// ---- POUs/Target/FB_PID.TcPOU
FUNCTION_BLOCK FB_PID
VAR_INPUT
	fSetpointValue: LREAL:=0;
	fActualValue :LREAL :=0;
	fFF:LREAL:=0;
	fKp: LREAL:=0;
	fKi: LREAL:=0;
	fKd: LREAL:=0;
	fKff: LREAL:=0;
	fIOutputMin: LREAL:=0;
	fIOutputMax: LREAL:=0;
	fOutputMin:LREAL:=0;
	fOutputMax:LREAL:=0;
	bReset:BOOL:=FALSE;
END_VAR
VAR_OUTPUT
	fCtrlOutput: LREAL;
END_VAR
VAR
	fOutputFF:LREAL:=0;
    fOutputP:LREAL:=0;
	fOutputI:LREAL:=0;
	fOutputD:LREAL:=0;
	fError:LREAL:=0;
	fErrorOld:LREAL:=0;
END_VAR

// Function: Simple PID controller with FF and limits for integral..
// Custom implementation needed since integral high and low limits are 
// needed in order to prvent integral windup.
// Author: Anders Sandström 20200115
 
IF bReset THEN
  fOutputP:=0;
  fOutputI:=0;
  fOutputD:=0;
  fFF:=0;
  fCtrlOutput:=0;
  RETURN;
END_IF

fErrorOld := fError;
fError    := fActualValue-fSetpointValue;

fOutputFF := fFF*fKff;         
fOutputP  := fKp*fError;
fOutputI  := fOutputI + fKi* fError;
// Prevent integral windup
IF fOutputI > fIOutputMax THEN
  fOutputI := fIOutputMax;
ELSIF fOutputI < fIOutputMin THEN
  fOutputI := fIOutputMin; 
END_IF

fOutputD  :=  (fError-fErrorOld)*fKd;

fCtrlOutput := fOutputP + fOutputI + fOutputD + fOutputFF;
IF fCtrlOutput < fOutputMin THEN
  fCtrlOutput := fOutputMin;
ELSIF fCtrlOutput > fOutputMax THEN
  fCtrlOutput := fOutputMax;
END_IF

END_FUNCTION_BLOCK

// ---- POUs/Target/FB_PWM.TcPOU
FUNCTION_BLOCK FB_PWM
VAR_INPUT
	En: BOOL;
	bEnable: BOOL;                  // Enable PWM alg
	iBlockSampleTimeMicroS: DINT;   // How often this block is called 
	iProcessSampleTimeMicroS: DINT; // Pwm cycle time. iProcessSampleTimeMicroS >> iBlockSampleTimeMicroS to get a good PWM resolution
 	iDecimalPoint: INT;             // At which decimal should teh pwm take place
	fInput: LREAL;                  // Input process value (that will be PWM:ed) 
	// PWM type:
	// Optimized: The low and high values are as ebenly distibuted in time as possible
	// Simple:    Either the low or high values are output first then the other (depending on bPromoteHigh bit)
	ePwmType:E_PWM_TYPE:=E_PWM_TYPE.OPTIMIZED;  
	bPromoteHigh:BOOL:=TRUE; // Only used in simple mode.
END_VAR
VAR_OUTPUT
	EnO: BOOL;
	fOutput: LREAL;
	fOutputError:LREAL:=0;  // Esitmated error of the PWM alg.
END_VAR
VAR
	iNumCycles: DINT;
	iBase: DINT;
	fDecimals: LREAL;
	i: INT;
	iDecimalGain: DINT;
	fOutputHigh: LREAL;
	iHighCycles: DINT;
	iLowCycles: DINT;
	fOutputLow: LREAL;
	iCycleCounter: DINT;
	iLowCounter: INT;
	iHighCounter: INT;
	fActualPWM: LREAL;
	fSetpointPWM: LREAL;
	fInputOld:LREAL:=0;
END_VAR

// Function: PWM block to be used to enhance resolution of signals
//
// Usefull for instance when a ethercat slave communicates with ints and you need 
// higher precision than the int provides. The desired input value are then PWM so that the
// average over processSampleTime is as close as possile to the desired value.
// Block can execute in three different modes:
//   OPTIMIZED: The low and high values are as evently as possible distributed over time
//   SIMPLE:    All high or low values are output first then the other (depending on bPromoteHigh bit)
//   NONE:      Output is same as input (no PWM)
//
// Note: Average resolution will be higher on the cost of sample rate
// Note: Error of PWM alg can be seen in fOutputError
//
// Example: fInput = 23.33333333, iDecimalpoint=3  ==>
//            fOutput will be pulse width modulated with the two discrete values: 23.333 and 23.334
//            in 33% of iProcessSampleTimeMicroS fOutput will be 23.333 and
//            in 67% of iProcessSampleTimeMicroS fOutput will be 23.334
//
// Author: Anders Sandström 2018
//
IF bEnable THEN
  IF(fInput<>fInputOld) THEN // New input value
    iNumCycles:=iProcessSampleTimeMicroS/iBlockSampleTimeMicroS; //71 if 71ms and 1ms
	iDecimalGain:=1;
	FOR i:=1 TO iDecimalPoint DO
      iDecimalGain:=iDecimalGain*10; //10000 if iDecimalpoint is 4
	END_FOR
	iBase:=TRUNC(fInput*iDecimalGain); //=900004 if fOverride=90.00045
    fDecimals:=fInput*iDecimalGain-iBase; //=0.5 if fOverride=90.00045
	iHighCycles:=LREAL_TO_INT(iNumCycles*fDecimals);
    iLowCycles:=iNumCycles-iHighCycles;
    fOutputLow:=DINT_TO_LREAL(iBase)/iDecimalGain; //90.0004
    fOutputHigh:=DINT_TO_LREAL(iBase+1)/iDecimalGain; //90.0005
	iCycleCounter:=0;
	iLowCounter:=0;
	iHighCounter:=0;
	fOutputError:=(fDecimals-DINT_TO_LREAL(iHighCycles)/DINT_TO_LREAL(iNumCycles))/iDecimalGain;
	fSetpointPWM:=DINT_TO_LREAL(iHighCycles)/DINT_TO_LREAL(iLowCycles+iHighCycles);
    END_IF

    IF iCycleCounter > iNumCycles THEN
	  iCycleCounter:=0;
	  iLowCounter:=0;
	  iHighCounter:=0;	
    END_IF
    iCycleCounter:=iCycleCounter+1;
	
  CASE ePwmType OF
	E_PWM_TYPE.OPTIMIZED:  // Distribute low and high evenly in time
       IF iLowCycles > 0 THEN
	     IF iHighCycles > 0 THEN
	       //Both high and low should be output during the period
	       IF iLowCounter = 0 THEN
		     fOutput:=fOutputLow;
		     iLowCounter:=iLowCounter+1;
	       ELSE
	         IF iHighCounter = 0 THEN
		       fOutput:=fOutputHigh;
		       iHighCounter:=iHighCounter+1;
	         ELSE //both counters is atleast 1
		       fActualPWM:= DINT_TO_LREAL(iHighCounter)/DINT_TO_LREAL(iLowCounter+iHighCounter);
		       IF fActualPWM>fSetpointPWM THEN
		         fOutput:=fOutputLow;
		         iLowCounter:=iLowCounter+1;
		       ELSE
                 fOutput:=fOutputHigh;
		         iHighCounter:=iHighCounter+1;
		       END_IF				
	        END_IF				
	      END_IF
        ELSE		
	      fOutput:=fOutputLow;
	      iLowCounter:=iLowCounter+1;
        END_IF
      ELSE
        fOutput:=fOutputHigh;
	    iHighCounter:=iHighCounter+1;
      END_IF
	  
    E_PWM_TYPE.SIMPLE:  // Take all low or high first then the other
	  IF bPromoteHigh THEN  // All high first
        IF iHighCounter < iHighCycles THEN
          iHighCounter:=iHighCounter+1;
		  fOutput:=fOutputHigh;
		ELSE
		  iLowCounter:=iLowCounter+1;
		  fOutput:=fOutputLow;
        END_IF
	  ELSE                  // All low first
        IF iLowCounter < iLowCycles THEN
          iLowCounter:=iLowCounter+1;
		  fOutput:=fOutputLow;
		ELSE
		  iHighCounter:=iHighCounter+1;
		  fOutput:=fOutputHigh;
        END_IF
		  
	  END_IF
	E_PWM_TYPE.NONE:    // Output same as input
	  fOutput:=fInput;
	  iCycleCounter:=0;
	  iLowCounter:=0;
	  iHighCounter:=0;	
	END_CASE
    
ELSE	
	fOutput:=fInput;	
END_IF
fInputOld:=fInput;

END_FUNCTION_BLOCK

// ---- POUs/Target/FB_RampVelo.TcPOU
FUNCTION_BLOCK FB_RampVelo
VAR_INPUT
	bExecute:BOOL;
	fVelSetIn:LREAL:=0;
	iBlockSampleTimeMicroS:INT:=10000;
	fVelActIn:LREAL:=0;
END_VAR
VAR_IN_OUT
    fVelSetOut:LREAL:=0;
END_VAR
VAR
  fChangePerCycle:LREAL:=0;
  fCurrAcc:LREAL:=0;
  fAccX1:LREAL:=0.8;
  fAccX2:LREAL:=0.99;
  fAccY1:LREAL:=GVL_Parameters.fAccDefaultVel;
  fAccY2:LREAL:=GVL_Parameters.fAccDefaultVel*0.1;
  fAccK:LREAL:=0;
  fAccM:LREAL:=0;
  x:LREAL:=0;
  bExecuteOld:BOOL:=FALSE;
  fActVeloOld:LREAL:=0;  // Used for extra sanity check of velo
END_VAR

// Function: Ramp velocity with a defined acceleration.
// Accelerartion is ramped down when approaching velocity setpoint in order to reduce
// overshoot and oscillations..
// Author: Anders Sandström 20200114

IF NOT bExecute OR ABS(fVelSetIn) > GVL_Parameters.fMaximumSPeedSPRpm THEN
  fVelSetOut:=0;
  bExecuteOld:=bExecute;
  fActVeloOld:=fVelActIn;
  RETURN;
END_IF;

// Start at current velocity if retreigger (avoid go to zero)
IF NOT bExecuteOld AND bExecute THEN
  // Sanity check of the actual velocity
  IF fVelActIn > -GVL_Parameters.fMaximumSPeedRpm AND 
	 fVelActIn < GVL_Parameters.fMaximumSPeedRpm AND 
	 fActVeloOld > -GVL_Parameters.fMaximumSPeedRpm AND 
	 fActVeloOld < GVL_Parameters.fMaximumSPeedRpm THEN
	fVelSetOut:=(fVelActIn+fActVeloOld)/2;  //Set to average of two cycles
    
	//Ensure minimum velo setpoint positive  to allow smooth start (with high ff tourqe at start)
	IF fVelSetIn > 0 AND ABS(fVelSetOut) < GVL_Parameters.fMinVelSetpointAbsRpm THEN
		fVelSetOut:=GVL_Parameters.fMinVelSetpointAbsRpm;
	END_IF
	//Ensure minimum velo setpoint negative to allow smooth start (with high ff tourqu at start)
	IF fVelSetIn < 0 AND ABS(fVelSetOut) < GVL_Parameters.fMinVelSetpointAbsRpm THEN
		fVelSetOut:=-GVL_Parameters.fMinVelSetpointAbsRpm;
	END_IF
  ELSE
    fVelSetOut:=0;
  END_IF  
END_IF
bExecuteOld:=bExecute;
fActVeloOld:=fVelActIn;

IF fVelSetOut=fVelSetIn THEN
  fVelSetOut:=fVelSetIn;
  RETURN;
END_IF;

//Reduce overshoot by lowering acc when closing in on setpoint (linear)
//           Acceleration [rpm/s^2]
//                 ^
//  y1=defAcc     -|-----------------\
//                 |                  \  
//                 |                   \
//                 |                    \ 
//                 |                     \
//  y2=defAcc*0.1 -|                      \-----------------
//                 |--------------------------------------------> fSetOut/fSetIn []
//                                 x1=0.8 x2=1.0 

fAccK:=(fAccY2-fAccY1)/(fAccX2-fAccX1);
fAccM:= fAccY1-fAccK*fAccX1;
IF fVelSetIn<>0 THEN
  x:=fVelSetOut/fVelSetIn;
ELSE
  x:=1.0;
END_IF
// try linear ramp down off acceleration from 0.8*velsetin to velset in (from defacc to 0.1* defacc)
fCurrAcc:=GVL_Parameters.fAccDefaultVel;
IF fVelSetIn > fVelSetOut THEN 
  IF x > fAccX1 AND x <= fAccX2 AND fVelSetOut<fVelSetIn THEN
    fCurrAcc:=fAccK*fVelSetOut/fVelSetIn+fAccM;
  ELSIF x >= fAccX2 THEN
    fCurrAcc:=GVL_Parameters.fAccDefaultVel*0.1;
  END_IF
END_IF

// Change per execution
fChangePerCycle:=fCurrAcc/(1E6/iBlockSampleTimeMicroS);

// Ramp finished
IF ABS(fVelSetIn-fVelSetOut)<fChangePerCycle THEN
  fVelSetOut:=fVelSetIn;
  RETURN;
END_IF

//Acc
IF fVelSetIn > fVelSetOut THEN             // Acc
  fVelSetOut:=fVelSetOut+fChangePerCycle;
ELSIF fVelSetIn < fVelSetOut THEN          // Dec
  fVelSetOut:=fVelSetOut-fChangePerCycle;
END_IF

END_FUNCTION_BLOCK

// ---- POUs/Target/FB_ModeVelo.TcPOU
FUNCTION_BLOCK FB_ModeVelo
VAR_INPUT
	bExecute:BOOL;
	bReset: BOOL;
	fVelSet:LREAL:=0;
	stStatus: ST_INDRADRIVE_AXIS_STATUS;
END_VAR
VAR_OUTPUT
	fSpeedSetpoint:LREAL:=0;
	bError: BOOL;
	nErrorId: UDINT;
	sErrorStr: STRING:=GVL_ErrorCodes.nErrorCodeOKStr;
END_VAR
VAR_IN_OUT
	stCommands: ST_INDRADRIVE_AXIS_COMMAND;
END_VAR

// Function: Constant velocity of target main  motor
// Control will be performed by the drive.
// Author: Anders Sandström 2018

stCommands.eMotionMode :=e_Motion_mode.eJogPositive;
stCommands.eOperationMode:=e_Operation_mode_no.eSecondaryOpMode2;
IF bExecute THEN
	fSpeedSetpoint:=fVelSet;
ELSE
	fSpeedSetpoint:=0;
END_IF
stCommands.fCommandVelocity:=0; // Other mode

END_FUNCTION_BLOCK

// ---- POUs/Target/FB_ModePos.TcPOU
FUNCTION_BLOCK FB_ModePos
VAR_INPUT
	bExecute:BOOL;
	bReset: BOOL;
	fVelSet:LREAL:=0;
	fPosSet:LREAL:=0;
	fRefOffset:LREAL:=0;  //Offset from homing
	stStatus: ST_INDRADRIVE_AXIS_STATUS;
END_VAR
VAR_OUTPUT
	bError: BOOL;
	nErrorId: UDINT;
	sErrorStr: STRING:=GVL_ErrorCodes.nErrorCodeOKStr;
END_VAR
VAR_IN_OUT
	stCommands: ST_INDRADRIVE_AXIS_COMMAND;
END_VAR
VAR
	fActPos:LREAL:=0;
    bExecuteOld:BOOL:=FALSE;
    //fPosSetTemp:LREAL:=0;
	fDistToTarget:LREAL:=0;
	//fDistToTrajSet:LREAL:=0;
	bVeloMode:BOOL:=FALSE;
END_VAR

// Function: Absolute positioning of target main  motor
// Actual positioning will be performed by the drive.
// Author: Anders Sandström 2018

stCommands.eMotionMode :=e_Motion_mode.ePositioning;
stCommands.eOperationMode:=e_Operation_mode_no.ePrimaryOpMode;
//stCommands.eOperationMode:=e_Operation_mode_no.eSecondaryOpMode3;

fActPos:=stStatus.fActualPosition-fRefOffset;
IF fActPos > 360 THEN
  fActPos:=fActPos-360;	
END_IF
IF fActPos < 0 THEN
  fActPos:=fActPos+360;	
END_IF

fDistToTarget:=FC_DistMod(fPosFrom:=fActPos,fPosTo:=fPosSet,fModRange:=360);
IF bExecute AND  NOT bExecuteOld THEN
  IF ABS(fDistToTarget) > 30 THEN   
    bVeloMode:=TRUE;
  ELSE
    bVeloMode:=FALSE;	 
  END_IF
END_IF

IF NOT bExecute THEN
  bVeloMode:=FALSE;
END_IF;	 
IF bExecute THEN
  IF bVeloMode THEN
	IF fDistToTarget> 0 THEN
	  stCommands.fVelocityCommandValue:=fVelSet;
	  IF fDistToTarget>0 THEN
	    stCommands.eMotionMode :=e_Motion_mode.eJogPositive;
	  ELSE
		 stCommands.eMotionMode :=e_Motion_mode.eJogNegative;
	  END_IF
      stCommands.eOperationMode:=e_Operation_mode_no.eSecondaryOpMode2;
	END_IF
	IF ABS(fDistToTarget) < 30 THEN 
		stCommands.fVelocityCommandValue:=0;
		IF stStatus.fActualVelocity <  fVelSet THEN
			bVeloMode:=FALSE;
		END_IF
	END_IF
  ELSE   // positioning
      stCommands.fCommandPosition:=fPosSet + fRefOffset;
      IF stCommands.fCommandPosition > 360 THEN
        stCommands.fCommandPosition:=stCommands.fCommandPosition-360;	
      END_IF
      IF stCommands.fCommandPosition < 0 THEN
         stCommands.fCommandPosition:=stCommands.fCommandPosition+360;	
      END_IF
      stCommands.fCommandVelocity:=fVelSet;
	  stCommands.eMotionMode :=e_Motion_mode.ePositioning;
      stCommands.eOperationMode:=e_Operation_mode_no.ePrimaryOpMode;
	  stCommands.fVelocityCommandValue:=0;
  END_IF
ELSE  
  stCommands.fCommandVelocity:=0;
  stCommands.fVelocityCommandValue:=0;
END_IF


//fDistToTrajSet:=FC_DistMod(fPosFrom:=fActPos,fPosTo:=fPosSetTemp,fModRange:=360);


(*IF ABS(fDistToTrajSet) < GVL_Parameters.fReachedTol THEN
  IF fDistToTarget > 0 THEN  // Increase traj setpoint with one step
	  fPosSetTemp:= fPosSetTemp + GVL_Parameters.fPosStep;
  ELSE
	  fPosSetTemp:= fPosSetTemp - GVL_Parameters.fPosStep;
  END_IF
END_IF

IF ABS(fDistToTarget) < GVL_Parameters.fPosStep THEN
   fPosSetTemp:=fPosSet;
END_IF

IF bExecute THEN
  stCommands.fCommandPosition:=fPosSetTemp + fRefOffset;
  IF stCommands.fCommandPosition > 360 THEN
    stCommands.fCommandPosition:=stCommands.fCommandPosition-360;	
  END_IF
  IF stCommands.fCommandPosition < 0 THEN
    stCommands.fCommandPosition:=stCommands.fCommandPosition+360;	
  END_IF
  stCommands.fCommandVelocity:=fVelSet;
ELSE
  stCommands.fCommandPosition:=stStatus.fActualPosition;
  stCommands.fCommandVelocity:=0;
END_IF*)


//stCommands.fVelocityCommandValue:=0;  //Used for other mode
bExecuteOld:=bExecute;

END_FUNCTION_BLOCK

// ---- POUs/Target/FB_ModeHome.TcPOU
FUNCTION_BLOCK FB_ModeHome
VAR_INPUT
	bExecute           : BOOL  := FALSE;
	bReset             : BOOL  := FALSE;
	fVelSet            : LREAL := 0;
	fPosSet            : LREAL := 0;
	stStatus           : ST_INDRADRIVE_AXIS_STATUS;
END_VAR
VAR_OUTPUT
	fSpeedSetpoint     : LREAL  := 0;
	fActPositionOffset : LREAL  := 0;
	bBusy              : BOOL   := FALSE;
	bError             : BOOL   := 0;
	nErrorId           : UDINT  := 0;
	sErrorStr          : STRING := GVL_ErrorCodes.nErrorCodeOKStr;
END_VAR
VAR_IN_OUT
	stCommands : ST_INDRADRIVE_AXIS_COMMAND;
	bHomed     : BOOL;
END_VAR
VAR
  bRefMarkPosArrayConsistent : BOOL  := FALSE;
  bTriggLatchMark            : BOOL  := FALSE;
  bExecuteOld                : BOOL  := FALSE;  
  nRevCounter                : UDINT := 0;
  nCounter                   : UDINT := 0;
  nRefMarksTotCount          : UDINT := 0;
  i                          : UDINT := 0;
  fNewestRefMarkPos          : LREAL := 0;
  fActPosAtHomeStart         : LREAL := 0;
  fMarkerPositionOld         : LREAL := 0;
  fActPositionOld            : LREAL := 0;
  fRefMarkPosArray           : ARRAY[ 0 ..GVL_Parameters.nRefMarkArraySize] OF LREAL;
  eHomeState                 : E_HOME_STATE := E_HOME_STATE.IDLE;
END_VAR

// Function: Initiate homing of target main motor
// Homing procedure:
// 1. Ramp up to (95% of) homing velocity (GVL_Parameters.fHomeSpeedRpm)
// 2. Issue drive command C1400 (latch encoder mark position)
//    - Latch GVL_Parameters.nRefMarkArraySize times (revolutions).
//    - Check that one latch per rev occurs.
//    - Check that all the latched psoitions are same.
//    - If everything is OK then store the position offset in fActPositionOffset 
//    - and set the bHomed flag. 
// 3. Ramp down.
// 4. Homing procedure is finalized
//    Now the fActPositionOffset can be used to offset the position from the drive
//    bBusy is set to false.
//
// Note: Homing is here in TwinCAT since the built in homing procedure cannot be used since
//       position loop in the drive is imposible to tune. 
//       This procedure runs the motor in velocity mode which are used for all other modes 
//       and can be releatively well tuned.
//
// Author: Anders Sandström 2018
//

// Test to ref in const velo
stCommands.eMotionMode :=e_Motion_mode.eJogPositive;
stCommands.eOperationMode:=e_Operation_mode_no.eSecondaryOpMode2;
stCommands.bCmd_NCHomeEnable:=TRUE;  // not used
stCommands.fCommandVelocity:=0; // Other mode
stCommands.bCmd_GetMarkerPosition:=bTriggLatchMark;
// Clear array and start
IF NOT bExecute AND eHomeState <> E_HOME_STATE.IDLE THEN
  eHomeState:=E_HOME_STATE.RAMP_DOWN;
END_IF

IF bReset THEN
  bError    := FALSE;
  nErrorID  := 0;
  sErrorStr := GVL_ErrorCodes.nErrorCodeOKStr;	
END_IF

CASE eHomeState OF
  E_HOME_STATE.IDLE:
    bBusy:=FALSE;
    IF bExecute AND NOT bExecuteOld AND NOT bError THEN
	  // Clear buffer and reset variables on state transition
      MEMSET(ADR(fRefMarkPosArray),0,SIZEOF(fRefMarkPosArray));
	  bBusy              := TRUE;  
      bTriggLatchMark    := FALSE;
      bHomed             := FALSE;
      nRefMarksTotCount  := 0;
	  nRevCounter        := 0;
	  fSpeedSetpoint     := 0;
	  fActPosAtHomeStart := 0;
	  fActPositionOffset := 0;
	  fNewestRefMarkPos  := 0;
	  eHomeState:=E_HOME_STATE.RAMP_UP;
    END_IF

  E_HOME_STATE.RAMP_UP:
    // Wait until reached velocity (once)
	fSpeedSetpoint:=fVelSet;
	bBusy:=TRUE;
    IF stStatus.fActualVelocity/10 > 0.95 * GVL_Parameters.fHomeSpeedRpm THEN
	  fActPosAtHomeStart := stStatus.fActualPosition;
      eHomeState:=E_HOME_STATE.HOMING;
	  bTriggLatchMark := TRUE;
    END_IF
	
  E_HOME_STATE.HOMING:
    // Move new latched value to buffer (newest always on index 0)
    IF (*stStatus.bCmd_GetMarkerPositionDone*) fMarkerPositionOld <> stStatus.fMarkerPosition AND 
      stStatus.fMarkerPosition <> 0 THEN
      MEMMOVE(ADR(fRefMarkPosArray)+SIZEOF(LREAL),ADR(fRefMarkPosArray),SIZEOF(fRefMarkPosArray)-SIZEOF(LREAL));
      fRefMarkPosArray[0]:=stStatus.fMarkerPosition;
      nCounter:=0;
      nRefMarksTotCount:=nRefMarksTotCount+1;
      // Check that complete buffer have same value (same latched value for all revs)
      IF nRefMarksTotCount >= GVL_Parameters.nRefMarkArraySize THEN
        fNewestRefMarkPos:=fRefMarkPosArray[0];
        bRefMarkPosArrayConsistent := TRUE;
        FOR i:=1 TO GVL_Parameters.nRefMarkArraySize - 1 DO
	      IF bRefMarkPosArrayConsistent THEN
	        bRefMarkPosArrayConsistent := fRefMarkPosArray[i] = fNewestRefMarkPos;
	      END_IF
        END_FOR
        bHomed:=bRefMarkPosArrayConsistent;
		IF bHomed THEN
		  fActPositionOffset := fNewestRefMarkPos+GVL_Parameters.fRotPosOffsetDeg;
		  IF fActPositionOffset>360 THEN
			  fActPositionOffset:=fActPositionOffset-360;
		  END_IF
		  IF fActPositionOffset<0 THEN
			  fActPositionOffset:=360+fActPositionOffset;
		  END_IF
		  
		ELSE
		  bError:=TRUE;	
          nErrorId:=GVL_ErrorCodes.nErrorEncoderLatchMissMatch;
          sErrorStr:=GVL_ErrorCodes.sErrorEncoderLatchMissMatch; 
		END_IF
      END_IF
    END_IF

    // Wait 100 cycles to ensure communication with drive..
    IF stStatus.fMarkerPosition <> 0 AND nCounter > 100 THEN
      bTriggLatchMark:=NOT bTriggLatchMark;
      nCounter:=0;  // wait for "response"
    END_IF
    nCounter:=nCounter+1;
	
    // Count revs since start homing. Must be one latch per rev.
	IF stStatus.fActualPosition > fActPosAtHomeStart AND fActPositionOld <= fActPosAtHomeStart THEN
      nRevCounter := nRevCounter+1;
	END_IF
	
	IF nRevCounter - nRefMarksTotCount > 1 THEN
	  bError := TRUE;
	  nErrorID := GVL_ErrorCodes.nErrorEncoderLatchLost;
	  sErrorStr := GVL_ErrorCodes.sErrorEncoderLatchLost;
	  eHomeState := E_HOME_STATE.RAMP_DOWN;
	END_IF
	
	IF nRefMarksTotCount > GVL_Parameters.nRefMarkArraySize OR bError THEN
	  eHomeState := E_HOME_STATE.RAMP_DOWN;
	END_IF
	
  E_HOME_STATE.RAMP_DOWN:
    fSpeedSetpoint:=0;
	IF stStatus.bAxisStandStillStatus THEN
	  eHomeState:=E_HOME_STATE.IDLE;
	  bBusy:=FALSE;
	END_IF
	
  ELSE
	eHomeState:=E_HOME_STATE.RAMP_DOWN;	
	
END_CASE

fMarkerPositionOld:=stStatus.fMarkerPosition;
fActPositionOld := stStatus.fActualPosition;
bExecuteOld:=bExecute;

END_FUNCTION_BLOCK

// ---- POUs/Target/FB_CalcVeloFromLatch.TcPOU
FUNCTION_BLOCK FB_CalcVeloFromLatch
VAR_INPUT
    dLatchedPosition   : DINT         := 0;
	fVeloLimit         : LREAL        := 3;
END_VAR
VAR_OUTPUT
	bError             : BOOL;
	nErrorId           : UDINT;
	sErrorStr          : STRING := GVL_ErrorCodes.nErrorCodeOKStr;
	fSpeedActual       : LREAL;
END_VAR
VAR
  dLatchedPositionOld      : DINT  := 0;
  fLatchedPositionOld      : LREAL := 0;
  fDistBetweenLastPulses   : LREAL := 0;
  fLastSectorVelocity      : LREAL := 0;
  fLatchedPosition         : LREAL := 0;
  fLastSectorVelocityOld   : LREAL := 0;
 END_VAR

// Function: 
// Calc velocity from drive latched positions (latched by timing system).
// This will result in an average velocity (for each sector at nominal speed) updated at 14Hz
// Author: Anders Sandström 2022

fLatchedPositionOld:=fLatchedPosition;  // Backup old
fLatchedPosition:=DINT_TO_LREAL(dLatchedPosition)/10000.0;  // remove homing offset
IF fLatchedPosition > 360 THEN
  fLatchedPosition:=fLatchedPosition - 360;	
END_IF
IF fLatchedPosition < 0 THEN
  fLatchedPosition:=fLatchedPosition + 360;	
END_IF

// New trigger from timing system
IF (fLatchedPosition-fLatchedPositionOld)<>0 THEN
  
  fDistBetweenLastPulses:=fLatchedPosition-fLatchedPositionOld;
  // Check over/underflow
  IF (ABS(fLatchedPositionOld - fLatchedPosition) > 200 ) THEN
    IF(fLatchedPositionOld > fLatchedPosition) THEN
	  // overflow
	  fDistBetweenLastPulses:=(360 - fLatchedPositionOld+fLatchedPosition);
    ELSE
	  // underflow
	  fDistBetweenLastPulses:=  fLatchedPositionOld +  fLatchedPosition-360;  
    END_IF
  END_IF

  fLastSectorVelocity:=fDistBetweenLastPulses*GVL_Parameters.nPulseFreqHz*60/360;
  fLastSectorVelocityOld:=fLastSectorVelocity;
END_IF

dLatchedPositionOld:=dLatchedPosition;
fSpeedActual:=fLastSectorVelocity;

END_FUNCTION_BLOCK

// ---- POUs/Target/fbIndraDrive.TcPOU
FUNCTION_BLOCK fbIndraDrive
VAR_INPUT 
	AmsNetId			: AMSNETID;		// AMS Net Id of the EtherCAT Master
	AdsAddr_Port		: WORD; 		// EtherCAT address of the Drive
	stAxisCommands		: ST_INDRADRIVE_AXIS_COMMAND; 
	stDriveStatus		: ST_INDRADRIVE_IO_INPUT; 
END_VAR
VAR_OUTPUT
	stAxisStatus		: ST_INDRADRIVE_AXIS_STATUS; 
	stDriveCommands		: ST_INDRADRIVE_IO_OUTPUT; 
END_VAR
VAR
	sAmsNetId						: T_AmsNetId;
	fbReadParameter					: FB_EcSoERead;
	nS149_DataStatus				: UDINT	:= 0;
END_VAR

VAR CONSTANT
	cC1300_LimitsEnabled			: UDINT := 0;
	cC1300_LimitsDisableActivated	: UDINT := 7;
	cC1300_LimitsDisabled			: UDINT := 3;
END_VAR

//==================================================================================================
//====== FunctionBlock to manage IndraDrive status and command =====================================
//==================================================================================================

// Create the T_AmsNetId 
sAmsNetId := F_CreateAmsNetId(AmsNetId); 

(*==================================================================================================================================================
=============    STATUS FROM THE DRIVE    ==========================================================================================================
==================================================================================================================================================*)
	// Display Drive status
		// Drive parameter mode  
		stAxisStatus.bDriveInParameterMode			:= stDriveStatus.stS144_SignalStatusWord.bS424_DriveMode; 

		// Drive Operation mode number
		IF (NOT stDriveStatus.nS135_DriveStatusWord.bS135_ActualOperationMode_Bit2) AND (NOT stDriveStatus.nS135_DriveStatusWord.bS135_ActualOperationMode_Bit1) AND (NOT stDriveStatus.nS135_DriveStatusWord.bS135_ActualOperationMode_Bit0) THEN 
			stAxisStatus.eActualOperationModeNo	:= E_OPERATION_MODE_NO.ePrimaryOpMode; 
		ELSIF (NOT stDriveStatus.nS135_DriveStatusWord.bS135_ActualOperationMode_Bit2) AND (NOT stDriveStatus.nS135_DriveStatusWord.bS135_ActualOperationMode_Bit1) AND stDriveStatus.nS135_DriveStatusWord.bS135_ActualOperationMode_Bit0 THEN 
			stAxisStatus.eActualOperationModeNo	:= E_OPERATION_MODE_NO.eSecondaryOpMode1; 
		ELSIF (NOT stDriveStatus.nS135_DriveStatusWord.bS135_ActualOperationMode_Bit2) AND stDriveStatus.nS135_DriveStatusWord.bS135_ActualOperationMode_Bit1 AND (NOT stDriveStatus.nS135_DriveStatusWord.bS135_ActualOperationMode_Bit0) THEN 
			stAxisStatus.eActualOperationModeNo	:= E_OPERATION_MODE_NO.eSecondaryOpMode2; 
		ELSIF (NOT stDriveStatus.nS135_DriveStatusWord.bS135_ActualOperationMode_Bit2) AND stDriveStatus.nS135_DriveStatusWord.bS135_ActualOperationMode_Bit1 AND stDriveStatus.nS135_DriveStatusWord.bS135_ActualOperationMode_Bit0 THEN 
			stAxisStatus.eActualOperationModeNo	:= E_OPERATION_MODE_NO.eSecondaryOpMode3; 
		ELSIF stDriveStatus.nS135_DriveStatusWord.bS135_ActualOperationMode_Bit2 AND (NOT stDriveStatus.nS135_DriveStatusWord.bS135_ActualOperationMode_Bit1) AND (NOT stDriveStatus.nS135_DriveStatusWord.bS135_ActualOperationMode_Bit0) THEN 
			stAxisStatus.eActualOperationModeNo	:= E_OPERATION_MODE_NO.eSecondaryOpMode4; 
		ELSIF stDriveStatus.nS135_DriveStatusWord.bS135_ActualOperationMode_Bit2 AND (NOT stDriveStatus.nS135_DriveStatusWord.bS135_ActualOperationMode_Bit1) AND stDriveStatus.nS135_DriveStatusWord.bS135_ActualOperationMode_Bit0 THEN 
			stAxisStatus.eActualOperationModeNo	:= E_OPERATION_MODE_NO.eSecondaryOpMode5; 
		ELSIF stDriveStatus.nS135_DriveStatusWord.bS135_ActualOperationMode_Bit2 AND stDriveStatus.nS135_DriveStatusWord.bS135_ActualOperationMode_Bit1 AND (NOT stDriveStatus.nS135_DriveStatusWord.bS135_ActualOperationMode_Bit0) THEN 
			stAxisStatus.eActualOperationModeNo	:= E_OPERATION_MODE_NO.eSecondaryOpMode6; 
		ELSIF stDriveStatus.nS135_DriveStatusWord.bS135_ActualOperationMode_Bit2 AND stDriveStatus.nS135_DriveStatusWord.bS135_ActualOperationMode_Bit1 AND stDriveStatus.nS135_DriveStatusWord.bS135_ActualOperationMode_Bit0 THEN 
			stAxisStatus.eActualOperationModeNo	:= E_OPERATION_MODE_NO.eSecondaryOpMode7; 
		END_IF
		// DC Bus
		stAxisStatus.bDCBusPresent					:= (*(NOT stDriveStatus.nS135_DriveStatusWord.bS135_ReadyForOperation_Bit0) AND *) stDriveStatus.nS135_DriveStatusWord.bS135_ReadyForOperation_Bit1; 
		// Axis enabled 
		stAxisStatus.bAxisEnabled					:= stDriveStatus.nS135_DriveStatusWord.bS135_ReadyForOperation_Bit0 AND stDriveStatus.nS135_DriveStatusWord.bS135_ReadyForOperation_Bit1; 
		// Absolute position status
		stAxisStatus.bAxisHomedStatus				:= stDriveStatus.stS144_SignalStatusWord.bS403_0_AxisHomedStatus; 
		// Axis standstill status 
		stAxisStatus.bAxisStandStillStatus			:= stDriveStatus.stS144_SignalStatusWord.bS331_StandStillStatus; 
		// Axis in target position
		stAxisStatus.bAxisInTargetPosition			:= stDriveStatus.stS144_SignalStatusWord.bS437_2_CommandPositionReached;
 		// Axis in constant velocity
		stAxisStatus.bAxisConstantVelocityStatus	:= (NOT stDriveStatus.stS144_SignalStatusWord.bS331_StandStillStatus) AND (NOT stDriveStatus.stS144_SignalStatusWord.bS437_5_Acceleration) AND (NOT stDriveStatus.stS144_SignalStatusWord.bS437_6_Deceleration);
 		// Axis in Acceleration
		stAxisStatus.bAxisAccelerationStatus		:= stDriveStatus.stS144_SignalStatusWord.bS437_5_Acceleration;
 		// Axis in Deceleration
		stAxisStatus.bAxisDecelerationStatus		:= stDriveStatus.stS144_SignalStatusWord.bS437_6_Deceleration;
 		// Axis in Jog
		stAxisStatus.bAxisJogStatus					:= stDriveStatus.stS144_SignalStatusWord.bS437_12_JogMode;
		// Drive command change 
		stAxisStatus.bCommandChange					:= stDriveStatus.nS135_DriveStatusWord.bS135_CommandChange; 
		// Drive command value processing  
		stAxisStatus.bCommandValueProcessing		:= stDriveStatus.stS144_SignalStatusWord.bP115_3_StatusOfCmdValueProcessing; 
        // STO active  ch1        
        stAxisStatus.bSTOActiveCh1:= stDriveStatus.stS144_SignalStatusWord.bP106_1_STO_ch1;
		// STO active  ch2       
        stAxisStatus.bSTOActiveCh2:= stDriveStatus.stS144_SignalStatusWord.bP106_2_STO_ch2;
        // C1400 Get Marker Position
		stAxisStatus.bCmd_GetMarkerPositionDone     := stDriveStatus.stS144_SignalStatusWord.bP14_0_C1400_GetMarkerPositionDone;
		
		// Disable monitoring  
		IF 	(stAxisCommands.bCmd_DisableLimits AND (NOT stAxisStatus.bLimitsDisabled)) OR 
			((NOT stAxisCommands.bCmd_DisableLimits) AND stAxisStatus.bLimitsDisabled) THEN
				fbReadParameter(
					sNetId:= sAmsNetId, 
					nSlaveAddr:= AdsAddr_Port, 
					nIdn:= 149, 
					nElement:= 16#01, 
					nDriveNo:= 0, 
					bCommand:= FALSE, 
					pDstBuf:= ADR(nS149_DataStatus), 
					cbBufLen:= SIZEOF(nS149_DataStatus), 
					bExecute:= TRUE, 
					tTimeout:= , 
					bBusy=> , 
					bError=> , 
					nErrId=> ); 
				
				IF (NOT fbReadParameter.bBusy) AND (NOT fbReadParameter.bError) THEN 
					IF (nS149_DataStatus = cC1300_LimitsDisableActivated) OR (nS149_DataStatus = cC1300_LimitsDisabled) THEN 
						stAxisStatus.bLimitsDisabled	:= TRUE;
					ELSIF (nS149_DataStatus = cC1300_LimitsEnabled) THEN 
						stAxisStatus.bLimitsDisabled	:= FALSE;
					END_IF
					// Execute with FALSE
					fbReadParameter(bExecute:= FALSE);
				END_IF
				
				IF fbReadParameter.bError THEN 
					// Execute with FALSE
					fbReadParameter(bExecute:= FALSE);
				END_IF
		END_IF
		
		// Diagnostic message present 
		stAxisStatus.bDiagMessage					:= stDriveStatus.nS135_DriveStatusWord.bS135_Class3_Diag_Mess;  
		// Warning message present 
		stAxisStatus.bWarning						:= stDriveStatus.nS135_DriveStatusWord.bS135_Class2_Diag_Warn;  
		// Error message present 
		stAxisStatus.bError							:= stDriveStatus.nS135_DriveStatusWord.bS135_Class1_Diag_Err;  
		// Diagnostic message number 
		{attribute 'displaymode':='hexadecimal'} 
		stAxisStatus.nDiagMessage					:= stDriveStatus.nS390_DiagnosticMessageNumber;
		
		// Display motion actual values 
		// Actual position (scale by 10000) 
		stAxisStatus.fActualPosition		:= DINT_TO_LREAL(stDriveStatus.nS386_ActivePositionFeedbackValue) / 10000.0; 
		// Actual velocity (scale by 1000) 
		stAxisStatus.fActualVelocity		:= DINT_TO_LREAL(stDriveStatus.nS40_VelocityFeedbackValue) / 1000.0; 
		// Actual Torque (scale by 10) 
		stAxisStatus.fActualTorque			:= INT_TO_LREAL(stDriveStatus.nS84_TorqueFeedback) / 10.0; 
		// Actual position error (scale by 10000) 
		stAxisStatus.fPositionError		:= DINT_TO_LREAL(stDriveStatus.nS189_PositionError) / 10000.0; 
        // Command C1400: Incremental encoder marker position (scale by 10000).
		stAxisStatus.fMarkerPosition := DINT_TO_LREAL(stDriveStatus.nP173_MarkerPosition) / 10000.0; 
		
(*==================================================================================================================================================
=============    COMMANDS TO THE DRIVE    ==========================================================================================================
==================================================================================================================================================*)
 	// Transfer and possibly scale command to the drive 
		// Operation mode 	
 		IF stAxisCommands.eOperationMode = E_OPERATION_MODE_NO.ePrimaryOpMode THEN 
			stDriveCommands.stS134_MasterControlWord.bS134_CmdOperationMode_Bit0 := FALSE;
			stDriveCommands.stS134_MasterControlWord.bS134_CmdOperationMode_Bit1 := FALSE;
			stDriveCommands.stS134_MasterControlWord.bS134_CmdOperationMode_Bit2 := FALSE;
		ELSIF stAxisCommands.eOperationMode = E_OPERATION_MODE_NO.eSecondaryOpMode1 THEN 
			stDriveCommands.stS134_MasterControlWord.bS134_CmdOperationMode_Bit0 := TRUE;
			stDriveCommands.stS134_MasterControlWord.bS134_CmdOperationMode_Bit1 := FALSE;
			stDriveCommands.stS134_MasterControlWord.bS134_CmdOperationMode_Bit2 := FALSE;
		ELSIF stAxisCommands.eOperationMode = E_OPERATION_MODE_NO.eSecondaryOpMode2 THEN 
			stDriveCommands.stS134_MasterControlWord.bS134_CmdOperationMode_Bit0 := FALSE;
			stDriveCommands.stS134_MasterControlWord.bS134_CmdOperationMode_Bit1 := TRUE;
			stDriveCommands.stS134_MasterControlWord.bS134_CmdOperationMode_Bit2 := FALSE;
		ELSIF stAxisCommands.eOperationMode = E_OPERATION_MODE_NO.eSecondaryOpMode3 THEN 
			stDriveCommands.stS134_MasterControlWord.bS134_CmdOperationMode_Bit0 := TRUE;
			stDriveCommands.stS134_MasterControlWord.bS134_CmdOperationMode_Bit1 := TRUE;
			stDriveCommands.stS134_MasterControlWord.bS134_CmdOperationMode_Bit2 := FALSE;
		ELSIF stAxisCommands.eOperationMode = E_OPERATION_MODE_NO.eSecondaryOpMode4 THEN 
			stDriveCommands.stS134_MasterControlWord.bS134_CmdOperationMode_Bit0 := FALSE;
			stDriveCommands.stS134_MasterControlWord.bS134_CmdOperationMode_Bit1 := FALSE;
			stDriveCommands.stS134_MasterControlWord.bS134_CmdOperationMode_Bit2 := TRUE;
		ELSIF stAxisCommands.eOperationMode = E_OPERATION_MODE_NO.eSecondaryOpMode5 THEN 
			stDriveCommands.stS134_MasterControlWord.bS134_CmdOperationMode_Bit0 := TRUE;
			stDriveCommands.stS134_MasterControlWord.bS134_CmdOperationMode_Bit1 := FALSE;
			stDriveCommands.stS134_MasterControlWord.bS134_CmdOperationMode_Bit2 := TRUE;
		ELSIF stAxisCommands.eOperationMode = E_OPERATION_MODE_NO.eSecondaryOpMode6 THEN 
			stDriveCommands.stS134_MasterControlWord.bS134_CmdOperationMode_Bit0 := FALSE;
			stDriveCommands.stS134_MasterControlWord.bS134_CmdOperationMode_Bit1 := TRUE;
			stDriveCommands.stS134_MasterControlWord.bS134_CmdOperationMode_Bit2 := TRUE;
		ELSIF stAxisCommands.eOperationMode = E_OPERATION_MODE_NO.eSecondaryOpMode7 THEN 
			stDriveCommands.stS134_MasterControlWord.bS134_CmdOperationMode_Bit0 := TRUE;
			stDriveCommands.stS134_MasterControlWord.bS134_CmdOperationMode_Bit1 := TRUE;
			stDriveCommands.stS134_MasterControlWord.bS134_CmdOperationMode_Bit2 := TRUE;
		END_IF
		
		// Enabling of the Axis 
		IF (NOT stAxisCommands.bEnableAxis) THEN 
			stDriveCommands.stS134_MasterControlWord.bS134_DriveEnable	:= FALSE; 
			stDriveCommands.stS134_MasterControlWord.bS134_DriveOn		:= FALSE; 
			stDriveCommands.stS134_MasterControlWord.bS134_DriveHalt	:= FALSE; 
		ELSIF stAxisCommands.bEnableAxis AND (NOT stAxisCommands.bHaltAxis) THEN 
			stDriveCommands.stS134_MasterControlWord.bS134_DriveEnable	:= TRUE; 
			stDriveCommands.stS134_MasterControlWord.bS134_DriveOn		:= TRUE; 
			stDriveCommands.stS134_MasterControlWord.bS134_DriveHalt	:= FALSE; 
		ELSIF stAxisCommands.bEnableAxis AND stAxisCommands.bHaltAxis THEN 
			stDriveCommands.stS134_MasterControlWord.bS134_DriveEnable	:= TRUE; 
			stDriveCommands.stS134_MasterControlWord.bS134_DriveOn		:= TRUE; 
			stDriveCommands.stS134_MasterControlWord.bS134_DriveHalt	:= TRUE; 
		END_IF
		
		// Positioning, Jog or stop the axis 
		stDriveCommands.nS47_PositionCommandValue 	:= stDriveStatus.nS386_ActivePositionFeedbackValue;
		stDriveCommands.nS282_PositioningCommandValue 	:= stDriveStatus.nS386_ActivePositionFeedbackValue;
		CASE stAxisCommands.eMotionMode OF 
			E_MOTION_MODE.eStop: 
				stDriveCommands.stS145_SignalControlWord.bS346_1_PosCtrlWord_PosActivation	:= TRUE; 
				stDriveCommands.stS145_SignalControlWord.bS346_2_PosCtrlWord_PosActivation	:= TRUE;
                stDriveCommands.nS258_TargetPosition 		:= stDriveStatus.nS386_ActivePositionFeedbackValue;			
			E_MOTION_MODE.eJogPositive: 
				stDriveCommands.stS145_SignalControlWord.bS346_1_PosCtrlWord_PosActivation	:= TRUE; 
				stDriveCommands.stS145_SignalControlWord.bS346_2_PosCtrlWord_PosActivation	:= FALSE;
                stDriveCommands.nS258_TargetPosition 		:= stDriveStatus.nS386_ActivePositionFeedbackValue; 				
			E_MOTION_MODE.eJogNegative: 
				stDriveCommands.stS145_SignalControlWord.bS346_1_PosCtrlWord_PosActivation	:= FALSE; 
				stDriveCommands.stS145_SignalControlWord.bS346_2_PosCtrlWord_PosActivation	:= TRUE;
                stDriveCommands.nS258_TargetPosition 		:= stDriveStatus.nS386_ActivePositionFeedbackValue;				
			E_MOTION_MODE.ePositioning: 
				stDriveCommands.stS145_SignalControlWord.bS346_1_PosCtrlWord_PosActivation	:= FALSE; 
				stDriveCommands.stS145_SignalControlWord.bS346_2_PosCtrlWord_PosActivation	:= FALSE;
		        stDriveCommands.nS258_TargetPosition := LREAL_TO_DINT(10000.0 * stAxisCommands.fCommandPosition);
		END_CASE
		
		// Position command change 
		stDriveCommands.stS145_SignalControlWord.bS346_5_PosCtrlWord_ImmBlockChange	:= stAxisCommands.bCommandPositionChange; 
        
        // 282 drive controlled positioning
		// 258 "Drive-internal interpolat
		// 47: cyclic position setpoint
		// Command position depending on Operation mode
		
		(*IF stAxisStatus.nDiagMessage >= 16#C00A0102 AND stAxisStatus.nDiagMessage <= 16#C00A0105 THEN
			stDriveCommands.nS47_PositionCommandValue 	:= LREAL_TO_DINT(10000.0 * stAxisCommands.fCommandPosition);
			stDriveCommands.nS282_PositioningCommandValue 	:= stDriveStatus.nS386_ActivePositionFeedbackValue;
			stDriveCommands.nS258_TargetPosition 		:= stDriveStatus.nS386_ActivePositionFeedbackValue;
		ELSIF (stAxisStatus.nDiagMessage >= 16#C00A0150 AND stAxisStatus.nDiagMessage <= 16#C00A0153) OR stAxisStatus.nDiagMessage = 16#C00A0161 THEN 
			stDriveCommands.nS282_PositioningCommandValue := LREAL_TO_DINT(10000.0 * stAxisCommands.fCommandPosition);
			stDriveCommands.nS47_PositionCommandValue 	:= stDriveStatus.nS386_ActivePositionFeedbackValue;
			stDriveCommands.nS258_TargetPosition 		:= stDriveStatus.nS386_ActivePositionFeedbackValue;
		ELSIF (stAxisStatus.nDiagMessage >= 16#C00A0106 AND stAxisStatus.nDiagMessage <= 16#C00A0109) THEN 
			stDriveCommands.nS258_TargetPosition := LREAL_TO_DINT(10000.0 * stAxisCommands.fCommandPosition);
			stDriveCommands.nS47_PositionCommandValue 	:= stDriveStatus.nS386_ActivePositionFeedbackValue;
			stDriveCommands.nS282_PositioningCommandValue 	:= stDriveStatus.nS386_ActivePositionFeedbackValue;
		END_IF*)
		
		// Did not enter any of the above cases so need to set for positioning mode.
		stDriveCommands.nS47_PositionCommandValue 	:= LREAL_TO_DINT(10000.0 * stAxisCommands.fCommandPosition);
			
		// Look for ref mark (latch)
		stDriveCommands.stS145_SignalControlWord.bP14_0_C1400_GetMarkerPosition := stAxisCommands.bCmd_GetMarkerPosition;
		// External home enabled
		stDriveCommands.stS145_SignalControlWord.bS407_0_HomingEnbale:=stAxisCommands.bCmd_NCHomeEnable;
		// Target velocity 
		stDriveCommands.nS259_PositioningVelocity := LREAL_TO_UDINT(10000.0 * stAxisCommands.fCommandVelocity);
		
		// Target acceleration 
		stDriveCommands.nS260_PositioningAcceleration := LREAL_TO_UDINT(1000.0 * stAxisCommands.fCommandAcceleration);
		
		// Target deceleration 
		stDriveCommands.nS359_PositioningDeceleration := LREAL_TO_UDINT(1000.0 * stAxisCommands.fCommandDeceleration);

		// Feedrate override
		stDriveCommands.nS108_FeedrateOverride := LREAL_TO_UINT(100.0 * stAxisCommands.fFeedrateOverride);
		
		// Torque limit
		stDriveCommands.nS92_BiPolarTorqueLimit := LREAL_TO_INT(10.0 * stAxisCommands.fTorqueLimit);
		
		// Absolute or Relative target position values 
		stDriveCommands.stS145_SignalControlWord.bS346_3_PosCtrlWord_Abs_Rel := stAxisCommands.bPositionCommandValue;
		
		// Error reset 
		stDriveCommands.stS145_SignalControlWord.bS99_DriveErrorReset := stAxisCommands.bCmd_ErrorReset;
		
		// Set Absolute position 
		stDriveCommands.stS145_SignalControlWord.bP12_C300_SetAbsolutePosition := stAxisCommands.bCmd_SetAbsolutePosition;
		
		// Drive controlled homing
		stDriveCommands.stS145_SignalControlWord.bS148_C600_DriveControlledHoming := stAxisCommands.bCmd_DriveControlledHoming;

		// C1300 Disable monitoring command (in documentation called Positive Stop Drive Procedure) 
		stDriveCommands.stS145_SignalControlWord.bS159_C1300_Disable_Monitoring	:= stAxisCommands.bCmd_DisableLimits;

		// Activate parameter mode
		stDriveCommands.stS145_SignalControlWord.bS420_C0400_Activate_ParameterMode := stAxisCommands.bCmd_ActivateParameterMode;
		
		// Exit parameter mode
		stDriveCommands.stS145_SignalControlWord.bS422_C0200_Exit_ParameterMode := stAxisCommands.bCmd_ExitParameterMode;

		// Command value accept
		stDriveCommands.stS145_SignalControlWord.bS346_0_PosCtrlWord_CmdValueAccept := stAxisCommands.bCommandValueAccept; 
		
		stDriveCommands.nS40_VelocityCommandValue := LREAL_TO_UDINT(10000.0 * stAxisCommands.fVelocityCommandValue);

		// Run the Virtual Master
		IF stAxisCommands.bCmd_RunVirtualMater THEN 
			stDriveCommands.stS145_SignalControlWord.bP760_VM_PosCtrlWord_1_PosActivation	:= TRUE;
			//stDriveCommands.stS145_SignalControlWord.bP760_VM_PosCtrlWord_2_PosActivation	:= FALSE;
			stDriveCommands.stS145_SignalControlWord.bP760_VM_PosCtrlWord_CmdValueAccept	:= TRUE;
		ELSE
			stDriveCommands.stS145_SignalControlWord.bP760_VM_PosCtrlWord_1_PosActivation	:= TRUE;
			//stDriveCommands.stS145_SignalControlWord.bP760_VM_PosCtrlWord_2_PosActivation	:= TRUE;
			stDriveCommands.stS145_SignalControlWord.bP760_VM_PosCtrlWord_CmdValueAccept	:= FALSE;
		END_IF

END_FUNCTION_BLOCK

// ---- POUs/Common/Hardware/EtherCAT_Terminals/Digital_Inputs/EL1809.TcPOU
///EL1809 | HD EtherCAT Terminals, 16-channel digital input 24 V DC, 3 ms
FUNCTION_BLOCK EL1809

VAR_INPUT
    En              : BOOL;
    iTerminal_ID    : INT;
    ErrorSystem     : POINTER TO ST_ErrorSystem;
END_VAR

VAR_OUTPUT
    EnO                 : BOOL;
    bError              : BOOL;
	sErrorMessage       : STRING;
	bBI_1                AT %I*  : BOOL:=FALSE;
	bBI_2                AT %I*  : BOOL:=FALSE;
	bBI_3                AT %I*  : BOOL:=FALSE;
	bBI_4                AT %I*  : BOOL:=FALSE;
	bBI_5                AT %I*  : BOOL:=FALSE;
	bBI_6                AT %I*  : BOOL:=FALSE;
	bBI_7                AT %I*  : BOOL:=FALSE;
	bBI_8                AT %I*  : BOOL:=FALSE;
	bBI_9                AT %I*  : BOOL:=FALSE;
	bBI_10               AT %I*  : BOOL:=FALSE;
	bBI_11               AT %I*  : BOOL:=FALSE;
	bBI_12               AT %I*  : BOOL:=FALSE;
	bBI_13               AT %I*  : BOOL:=FALSE;
	bBI_14               AT %I*  : BOOL:=FALSE;
	bBI_15               AT %I*  : BOOL:=FALSE;
	bBI_16               AT %I*  : BOOL:=FALSE;
END_VAR

VAR
    WcState_WcState     AT %I*  : BOOL := TRUE;  // invalid
    InfoData_State      AT %I*  : UINT := 0;
    //dBI_all                     : INT  := 0;
    //FB-s
    EL1809_Error      : FB_TerminalError;
END_VAR

(*
* TODO: DONE!
*)
EnO:=En;
(*dBI_all.0:=bBI_1;
dBI_all.1:=bBI_2;
dBI_all.2:=bBI_3;
dBI_all.3:=bBI_4;
dBI_all.4:=bBI_5;
dBI_all.5:=bBI_6;
dBI_all.6:=bBI_7;
dBI_all.7:=bBI_8;
dBI_all.8:=bBI_9;
dBI_all.9:=bBI_10;
dBI_all.10:=bBI_11;
dBI_all.11:=bBI_12;
dBI_all.12:=bBI_13;
dBI_all.13:=bBI_14;
dBI_all.14:=bBI_15;
dBI_all.15:=bBI_16;*)

//Error FB instance
EL1809_Error(
    En                  := TRUE,
    iTerminal_ID        := iTerminal_ID,
    bWcState            := WcState_WcState,
    uiInfoData_State    := InfoData_State,
    pErrorSystem        := ErrorSystem,
    bError              => bError,
);

IF bError THEN
	sErrorMessage:=EL1809_Error.ErrorData.sErrorMessage;
ELSE
	sErrorMessage:='';
END_IF

END_FUNCTION_BLOCK

// ---- POUs/Common/ErrorHandling/FB_TerminalError.TcPOU
FUNCTION_BLOCK FB_TerminalError

VAR_INPUT
    En                  : BOOL;
    iTerminal_ID        : INT;
    bWcState            : BOOL;
    uiInfoData_State    : UINT;
    pErrorSystem        : POINTER TO ST_ErrorSystem;                    //Pointer to the error system
END_VAR

VAR_OUTPUT
    EnO : BOOL;
    bError : BOOL := FALSE;
END_VAR

VAR
    iStateError : UINT;
    iOtherError : UINT;
    ErrorData   : ST_ErrorEntry;
    nErrSysCNT  : UINT;

    bStateChanged           : BOOL;             //Indicate if state change happened
    uiInfoData_State_Prev   : UINT := 16#8;     //Previous value of Infodata.State
    bWcState_Prev           : BOOL := FALSE;    //Previous state of WcState

    //FB-s

END_VAR

(*
* ================================================================================
*                                   DESCRIPTION
* ================================================================================
* This Function Block provides connection to the Error System specifically
* for monitoring an EtherCat terminal's state of operation. The function block
* checks the content of the linked variables, that encodes the terminal's state.
* If any deviation from the nominal state is experienced an entry is created with
* all the necessary information. If the terminal goes through a series of
* different error states each state transition is tracked in a new entry.
* ================================================================================
*)

//Connect EN to EnO
EnO:=En;

IF En THEN
    //Check if pointer is OK
    IF pErrorSystem=0 THEN RETURN; END_IF

    //Any difference from normal state creates an error
    IF En AND (bWcState OR uiInfoData_State<>16#8) THEN
        bError:=TRUE;
    ELSE
        bError:=FALSE;
    END_IF

    //Change detection
    IF uiInfoData_State <> uiInfoData_State_Prev OR bWcState <> bWcState_Prev THEN
        bStateChanged := TRUE;
    ELSE
        bStateChanged := FALSE;
    END_IF

    //Update previous values
    uiInfoData_State_Prev   := uiInfoData_State;
    bWcState_Prev           := bWcState;

    //Decision tree
    IF bStateChanged THEN
        IF bError THEN
            IF ErrorData.ErrorState = DUT_ErrorState.Active THEN
                //Close active error
                //Read system time
                ErrorData.sDateTimeOff  := Tc2_EtherCat.DCTIME64_TO_STRING(Tc2_EtherCAT.F_GetActualDcTime64());
                ErrorData.ErrorState    := DUT_ErrorState.Inactive;
                //Write Off-time to Error System
                FOR nErrSysCNT := 0 TO cSizeOfErrorData - 1 DO
                    IF pErrorSystem^.aErrorData[nErrSysCNT].ErrorNum = ErrorData.ErrorNum THEN
                        pErrorSystem^.aErrorData[nErrSysCNT].sDateTimeOff   := ErrorData.sDateTimeOff;
                        pErrorSystem^.aErrorData[nErrSysCNT].ErrorState     := DUT_ErrorState.Inactive;
                        EXIT;
                    END_IF
                END_FOR

                //Clear ErrorData
                MEMSET(ADR(ErrorData), 0, SIZEOF(ErrorData));
            END_IF

            //Open a new error
            ErrorData.ErrorState    := DUT_ErrorState.Active;                                                   //Set Error State
            ErrorData.sDateTimeOn   := Tc2_EtherCat.DCTIME64_TO_STRING(Tc2_EtherCAT.F_GetActualDcTime64());     //Convert to string
            ErrorData.iTerminalID   := iTerminal_ID;                                                            //Terminal_ID

            //Error message according to uiInfoData_State and WcState
            iStateError := (uiInfoData_State AND 16#000F);                                              //Mask for operation state
            iOtherError := (uiInfoData_State AND 16#00F0);                                              //Mask for the other 3 kind of errors
            //Error messages according to the least significant digit
            CASE iStateError OF
                16#0001 :
                            ErrorData.sErrorMessage := 'Slave in INIT state;   ';
                            IF ErrorData.ErrorPriority >= 5 OR ErrorData.ErrorPriority = 0 THEN ErrorData.ErrorPriority := 5; END_IF
                16#0002 :
                            ErrorData.sErrorMessage := 'Slave in PREOP state;   ';
                            IF ErrorData.ErrorPriority >= 5 OR ErrorData.ErrorPriority = 0 THEN ErrorData.ErrorPriority := 5; END_IF
                16#0003 :
                            ErrorData.sErrorMessage := 'Slave in BOOT state;   ';
                            IF ErrorData.ErrorPriority >= 5 OR ErrorData.ErrorPriority = 0 THEN ErrorData.ErrorPriority := 5; END_IF
                16#0004 :
                            ErrorData.sErrorMessage := 'Slave in SAFEOP state;   ';
                            IF ErrorData.ErrorPriority >= 5 OR ErrorData.ErrorPriority = 0 THEN ErrorData.ErrorPriority := 5; END_IF
                16#0008 : ;                                                                             //Normal operation state
            ELSE
                ErrorData.sErrorMessage := 'Undefined State of operation;   ';
                ErrorData.sErrorMessage := CONCAT (ErrorData.sErrorMessage, UINT_TO_STRING(iStateError));
                ErrorData.sErrorMessage := CONCAT (ErrorData.sErrorMessage, '   ');
                ErrorData.ErrorPriority := 1;
            END_CASE

            //Error messages according to the second least significant digit
            CASE iOtherError OF
                16#0000 : ;                                                                         //No error case
                16#0010 :
                            ErrorData.sErrorMessage := CONCAT (ErrorData.sErrorMessage, 'Slave signals error;   ');
                            IF ErrorData.ErrorPriority >= 5 OR ErrorData.ErrorPriority = 0 THEN ErrorData.ErrorPriority := 5; END_IF
                16#0020 :
                            ErrorData.sErrorMessage := CONCAT (ErrorData.sErrorMessage, 'Invalid vendorID/productCode read;   ');
                            IF ErrorData.ErrorPriority >= 5 OR ErrorData.ErrorPriority = 0 THEN ErrorData.ErrorPriority := 5; END_IF
                16#0040 :
                            ErrorData.sErrorMessage := CONCAT (ErrorData.sErrorMessage, 'Initialisation error occured;   ');
                            IF ErrorData.ErrorPriority >= 5 OR ErrorData.ErrorPriority = 0 THEN ErrorData.ErrorPriority := 5; END_IF
            ELSE
                ErrorData.sErrorMessage := CONCAT (ErrorData.sErrorMessage, 'Undefined Error ID: ');
                ErrorData.sErrorMessage := CONCAT (ErrorData.sErrorMessage, UINT_TO_STRING(iOtherError));
                ErrorData.sErrorMessage := CONCAT (ErrorData.sErrorMessage, '   ');
                ErrorData.ErrorPriority := 1;
            END_CASE

            //Errormessage according to WcState bit
            IF bWcState THEN
                ErrorData.sErrorMessage := CONCAT (ErrorData.sErrorMessage, 'Invalid Data;');
                IF ErrorData.ErrorPriority >= 5 OR ErrorData.ErrorPriority = 0 THEN ErrorData.ErrorPriority := 5; END_IF
            END_IF

            //Check for overflow
            IF pErrorSystem^.nNoError >= cSizeOfErrorData THEN
                pErrorSystem^.nNoOverflow := pErrorSystem^.nNoOverflow+1;
            END_IF

            //Write Error Data into Error System
            ErrorData.ErrorNum  := pErrorSystem^.nNExtErrorNum ;
            MEMMOVE( ADR(pErrorSystem^.aErrorData[1]), ADR(pErrorSystem^.aErrorData[0]), (cSizeOfErrorData-1) * SIZEOF(ST_ErrorEntry));
            pErrorSystem^.aErrorData[0] := ErrorData;
            pErrorSystem^.nNExtErrorNum := pErrorSystem^.nNExtErrorNum+1;

        ELSE
            //Close Active Error
            //Read system time
            ErrorData.sDateTimeOff  := Tc2_EtherCat.DCTIME64_TO_STRING(Tc2_EtherCAT.F_GetActualDcTime64());
            ErrorData.ErrorState    := DUT_ErrorState.Inactive;
            //Write Off time to Error System
            FOR nErrSysCNT := 0 TO cSizeOfErrorData - 1 DO
                IF pErrorSystem^.aErrorData[nErrSysCNT].ErrorNum = ErrorData.ErrorNum THEN
                    pErrorSystem^.aErrorData[nErrSysCNT].sDateTimeOff   := ErrorData.sDateTimeOff;
                    pErrorSystem^.aErrorData[nErrSysCNT].ErrorState     := ErrorData.ErrorState;
                    EXIT;
                END_IF
            END_FOR

            //Clear ErrorData
            MEMSET(ADR(ErrorData), 0, SIZEOF(ErrorData));
        END_IF
    END_IF

END_IF

END_FUNCTION_BLOCK

// ---- POUs/Common/Hardware/EtherCAT_Terminals/Digital_Outputs/EL2819.TcPOU
FUNCTION_BLOCK EL2819
VAR_INPUT
    En              : BOOL;
    iTerminal_ID    : INT;
    ErrorSystem     : POINTER TO ST_ErrorSystem;
END_VAR

VAR_OUTPUT
    EnO     : BOOL;
    bError  : BOOL;
	sErrorMessage       : STRING;
END_VAR

VAR
    wCH1_Diag       AT %I*  : BYTE;
    wCH2_Diag       AT %I*  : BYTE;
    wCH3_Diag       AT %I*  : BYTE;
    wCH4_Diag       AT %I*  : BYTE;
    wCH5_Diag       AT %I*  : BYTE;
    wCH6_Diag       AT %I*  : BYTE;
    wCH7_Diag       AT %I*  : BYTE;
    wCH8_Diag       AT %I*  : BYTE;
    wCH9_Diag       AT %I*  : BYTE;
    wCH10_Diag      AT %I*  : BYTE;
    wCH11_Diag      AT %I*  : BYTE;
    wCH12_Diag      AT %I*  : BYTE;
    wCH13_Diag      AT %I*  : BYTE;
    wCH14_Diag      AT %I*  : BYTE;
    wCH15_Diag      AT %I*  : BYTE;
    wCH16_Diag      AT %I*  : BYTE;

    bDev_CommonFault            AT %I*  : BOOL;
    bDev_Overtemperature        AT %I*  : BOOL;
    bDev_UnderVoltage           AT %I*  : BOOL;
    bDev_MissingVoltage         AT %I*  : BOOL;

    WcState_WcState     AT %I*  : BOOL;
    InfoData_State      AT %I*  : UINT;

    //FB-s
    EL2819_Error    : FB_TerminalError;

    CH1_Error       : FB_GenericError;
    CH2_Error       : FB_GenericError;
    CH3_Error       : FB_GenericError;
    CH4_Error       : FB_GenericError;
    CH5_Error       : FB_GenericError;
    CH6_Error       : FB_GenericError;
    CH7_Error       : FB_GenericError;
    CH8_Error       : FB_GenericError;
    CH9_Error       : FB_GenericError;
    CH10_Error      : FB_GenericError;
    CH11_Error      : FB_GenericError;
    CH12_Error      : FB_GenericError;
    CH13_Error      : FB_GenericError;
    CH14_Error      : FB_GenericError;
    CH15_Error      : FB_GenericError;
    CH16_Error      : FB_GenericError;

    DEV_Error       : FB_GenericError;
END_VAR

(*
* TODO: test on hardware
*)

EnO:=En;

IF En THEN
    //Channel #1 Diag
    IF (wCH1_Diag AND 16#07) <> 0 THEN
        CH1_Error.sErrorMessage := 'EL2819 Channel #1: ';
        IF wCH1_Diag.0  THEN    CH1_Error.sErrorMessage := CONCAT(CH1_Error.sErrorMessage, 'Overtemperature; ');            IF CH1_Error.ErrorPriority > 10  OR CH1_Error.ErrorPriority = 0     THEN CH1_Error.ErrorPriority := 10;     END_IF      END_IF
        IF wCH1_Diag.1  THEN    CH1_Error.sErrorMessage := CONCAT(CH1_Error.sErrorMessage, 'Open Load; ');                  IF CH1_Error.ErrorPriority > 100 OR CH1_Error.ErrorPriority = 0     THEN CH1_Error.ErrorPriority := 100;    END_IF      END_IF
        IF wCH1_Diag.2  THEN    CH1_Error.sErrorMessage := CONCAT(CH1_Error.sErrorMessage, 'Overcurrent; ');                IF CH1_Error.ErrorPriority > 10  OR CH1_Error.ErrorPriority = 0     THEN CH1_Error.ErrorPriority := 10;     END_IF      END_IF
        IF wCH1_Diag.3  THEN    CH1_Error.sErrorMessage := CONCAT(CH1_Error.sErrorMessage, 'Short Circuit to 24V; ');       IF CH1_Error.ErrorPriority > 10  OR CH1_Error.ErrorPriority = 0     THEN CH1_Error.ErrorPriority := 10;     END_IF      END_IF
        CH1_Error.bError := TRUE;
    ELSE
        CH1_Error.bError := FALSE;
        CH1_Error.sErrorMessage := '';
    END_IF

    //Channel #2 Diag
    IF (wCH2_Diag AND 16#07) <> 0 THEN
        CH2_Error.sErrorMessage := 'EL2819 Channel #2: ';
        IF wCH2_Diag.0  THEN    CH2_Error.sErrorMessage := CONCAT(CH2_Error.sErrorMessage, 'Overtemperature; ');            IF CH2_Error.ErrorPriority > 10  OR CH2_Error.ErrorPriority = 0     THEN CH2_Error.ErrorPriority := 10;     END_IF      END_IF
        IF wCH2_Diag.1  THEN    CH2_Error.sErrorMessage := CONCAT(CH2_Error.sErrorMessage, 'Open Load; ');                  IF CH2_Error.ErrorPriority > 100 OR CH2_Error.ErrorPriority = 0     THEN CH2_Error.ErrorPriority := 100;    END_IF      END_IF
        IF wCH2_Diag.2  THEN    CH2_Error.sErrorMessage := CONCAT(CH2_Error.sErrorMessage, 'Overcurrent; ');                IF CH2_Error.ErrorPriority > 10  OR CH2_Error.ErrorPriority = 0     THEN CH2_Error.ErrorPriority := 10;     END_IF      END_IF
        IF wCH2_Diag.3  THEN    CH2_Error.sErrorMessage := CONCAT(CH2_Error.sErrorMessage, 'Short Circuit to 24V; ');       IF CH2_Error.ErrorPriority > 10  OR CH2_Error.ErrorPriority = 0     THEN CH2_Error.ErrorPriority := 10;     END_IF      END_IF
        CH2_Error.bError := TRUE;
    ELSE
        CH2_Error.bError := FALSE;
        CH2_Error.sErrorMessage := '';
    END_IF

    //Channel #3 Diag
    IF wCH3_Diag <> 0 THEN
        CH3_Error.sErrorMessage := 'EL2819 Channel #3: ';
        IF wCH3_Diag.0  THEN    CH3_Error.sErrorMessage := CONCAT(CH3_Error.sErrorMessage, 'Overtemperature; ');            IF CH3_Error.ErrorPriority > 10  OR CH3_Error.ErrorPriority = 0     THEN CH3_Error.ErrorPriority := 10;     END_IF      END_IF
        IF wCH3_Diag.1  THEN    CH3_Error.sErrorMessage := CONCAT(CH3_Error.sErrorMessage, 'Open Load; ');                  IF CH3_Error.ErrorPriority > 100 OR CH3_Error.ErrorPriority = 0     THEN CH3_Error.ErrorPriority := 100;    END_IF      END_IF
        IF wCH3_Diag.2  THEN    CH3_Error.sErrorMessage := CONCAT(CH3_Error.sErrorMessage, 'Overcurrent; ');                IF CH3_Error.ErrorPriority > 10  OR CH3_Error.ErrorPriority = 0     THEN CH3_Error.ErrorPriority := 10;     END_IF      END_IF
        IF wCH3_Diag.3  THEN    CH3_Error.sErrorMessage := CONCAT(CH3_Error.sErrorMessage, 'Short Circuit to 24V; ');       IF CH3_Error.ErrorPriority > 10  OR CH3_Error.ErrorPriority = 0     THEN CH3_Error.ErrorPriority := 10;     END_IF      END_IF
        CH3_Error.bError := TRUE;
    ELSE
        CH3_Error.bError := FALSE;
        CH3_Error.sErrorMessage := '';
    END_IF

    //Channel #4 Diag
    IF wCH4_Diag <> 0 THEN
        CH4_Error.sErrorMessage := 'EL2819 Channel #4: ';
        IF wCH4_Diag.0  THEN    CH4_Error.sErrorMessage := CONCAT(CH4_Error.sErrorMessage, 'Overtemperature; ');            IF CH4_Error.ErrorPriority > 10  OR CH4_Error.ErrorPriority = 0     THEN CH4_Error.ErrorPriority := 10;     END_IF      END_IF
        IF wCH4_Diag.1  THEN    CH4_Error.sErrorMessage := CONCAT(CH4_Error.sErrorMessage, 'Open Load; ');                  IF CH4_Error.ErrorPriority > 100 OR CH4_Error.ErrorPriority = 0     THEN CH4_Error.ErrorPriority := 100;    END_IF      END_IF
        IF wCH4_Diag.2  THEN    CH4_Error.sErrorMessage := CONCAT(CH4_Error.sErrorMessage, 'Overcurrent; ');                IF CH4_Error.ErrorPriority > 10  OR CH4_Error.ErrorPriority = 0     THEN CH4_Error.ErrorPriority := 10;     END_IF      END_IF
        IF wCH4_Diag.3  THEN    CH4_Error.sErrorMessage := CONCAT(CH4_Error.sErrorMessage, 'Short Circuit to 24V; ');       IF CH4_Error.ErrorPriority > 10  OR CH4_Error.ErrorPriority = 0     THEN CH4_Error.ErrorPriority := 10;     END_IF      END_IF
        CH4_Error.bError := TRUE;
    ELSE
        CH4_Error.bError := FALSE;
        CH4_Error.sErrorMessage := '';
    END_IF

    //Channel #5 Diag
    IF wCH5_Diag <> 0 THEN
        CH5_Error.sErrorMessage := 'EL2819 Channel #5: ';
        IF wCH5_Diag.0  THEN    CH5_Error.sErrorMessage := CONCAT(CH5_Error.sErrorMessage, 'Overtemperature; ');            IF CH5_Error.ErrorPriority > 10  OR CH5_Error.ErrorPriority = 0     THEN CH5_Error.ErrorPriority := 10;     END_IF      END_IF
        IF wCH5_Diag.1  THEN    CH5_Error.sErrorMessage := CONCAT(CH5_Error.sErrorMessage, 'Open Load; ');                  IF CH5_Error.ErrorPriority > 100 OR CH5_Error.ErrorPriority = 0     THEN CH5_Error.ErrorPriority := 100;    END_IF      END_IF
        IF wCH5_Diag.2  THEN    CH5_Error.sErrorMessage := CONCAT(CH5_Error.sErrorMessage, 'Overcurrent; ');                IF CH5_Error.ErrorPriority > 10  OR CH5_Error.ErrorPriority = 0     THEN CH5_Error.ErrorPriority := 10;     END_IF      END_IF
        IF wCH5_Diag.3  THEN    CH5_Error.sErrorMessage := CONCAT(CH5_Error.sErrorMessage, 'Short Circuit to 24V; ');       IF CH5_Error.ErrorPriority > 10  OR CH5_Error.ErrorPriority = 0     THEN CH5_Error.ErrorPriority := 10;     END_IF      END_IF
        CH5_Error.bError := TRUE;
    ELSE
        CH5_Error.bError := FALSE;
        CH5_Error.sErrorMessage := '';
    END_IF

    //Channel #6 Diag
    IF wCH6_Diag <> 0 THEN
        CH6_Error.sErrorMessage := 'EL2819 Channel #6: ';
        IF wCH6_Diag.0  THEN    CH6_Error.sErrorMessage := CONCAT(CH6_Error.sErrorMessage, 'Overtemperature; ');            IF CH6_Error.ErrorPriority > 10  OR CH6_Error.ErrorPriority = 0     THEN CH6_Error.ErrorPriority := 10;     END_IF      END_IF
        IF wCH6_Diag.1  THEN    CH6_Error.sErrorMessage := CONCAT(CH6_Error.sErrorMessage, 'Open Load; ');                  IF CH6_Error.ErrorPriority > 100 OR CH6_Error.ErrorPriority = 0     THEN CH6_Error.ErrorPriority := 100;    END_IF      END_IF
        IF wCH6_Diag.2  THEN    CH6_Error.sErrorMessage := CONCAT(CH6_Error.sErrorMessage, 'Overcurrent; ');                IF CH6_Error.ErrorPriority > 10  OR CH6_Error.ErrorPriority = 0     THEN CH6_Error.ErrorPriority := 10;     END_IF      END_IF
        IF wCH6_Diag.3  THEN    CH6_Error.sErrorMessage := CONCAT(CH6_Error.sErrorMessage, 'Short Circuit to 24V; ');       IF CH6_Error.ErrorPriority > 10  OR CH6_Error.ErrorPriority = 0     THEN CH6_Error.ErrorPriority := 10;     END_IF      END_IF
        CH6_Error.bError := TRUE;
    ELSE
        CH6_Error.bError := FALSE;
        CH6_Error.sErrorMessage := '';
    END_IF

    //Channel #7 Diag
    IF wCH7_Diag <> 0 THEN
        CH7_Error.sErrorMessage := 'EL2819 Channel #7: ';
        IF wCH7_Diag.0  THEN    CH7_Error.sErrorMessage := CONCAT(CH7_Error.sErrorMessage, 'Overtemperature; ');            IF CH7_Error.ErrorPriority > 10  OR CH7_Error.ErrorPriority = 0     THEN CH7_Error.ErrorPriority := 10;     END_IF      END_IF
        IF wCH7_Diag.1  THEN    CH7_Error.sErrorMessage := CONCAT(CH7_Error.sErrorMessage, 'Open Load; ');                  IF CH7_Error.ErrorPriority > 100 OR CH7_Error.ErrorPriority = 0     THEN CH7_Error.ErrorPriority := 100;    END_IF      END_IF
        IF wCH7_Diag.2  THEN    CH7_Error.sErrorMessage := CONCAT(CH7_Error.sErrorMessage, 'Overcurrent; ');                IF CH7_Error.ErrorPriority > 10  OR CH7_Error.ErrorPriority = 0     THEN CH7_Error.ErrorPriority := 10;     END_IF      END_IF
        IF wCH7_Diag.3  THEN    CH7_Error.sErrorMessage := CONCAT(CH7_Error.sErrorMessage, 'Short Circuit to 24V; ');       IF CH7_Error.ErrorPriority > 10  OR CH7_Error.ErrorPriority = 0     THEN CH7_Error.ErrorPriority := 10;     END_IF      END_IF
        CH7_Error.bError := TRUE;
    ELSE
        CH7_Error.bError := FALSE;
        CH7_Error.sErrorMessage := '';
    END_IF

    //Channel #8 Diag
    IF wCH8_Diag <> 0 THEN
        CH8_Error.sErrorMessage := 'EL2819 Channel #8: ';
        IF wCH8_Diag.0  THEN    CH8_Error.sErrorMessage := CONCAT(CH8_Error.sErrorMessage, 'Overtemperature; ');            IF CH8_Error.ErrorPriority > 10  OR CH8_Error.ErrorPriority = 0     THEN CH8_Error.ErrorPriority := 10;     END_IF      END_IF
        IF wCH8_Diag.1  THEN    CH8_Error.sErrorMessage := CONCAT(CH8_Error.sErrorMessage, 'Open Load; ');                  IF CH8_Error.ErrorPriority > 100 OR CH8_Error.ErrorPriority = 0     THEN CH8_Error.ErrorPriority := 100;    END_IF      END_IF
        IF wCH8_Diag.2  THEN    CH8_Error.sErrorMessage := CONCAT(CH8_Error.sErrorMessage, 'Overcurrent; ');                IF CH8_Error.ErrorPriority > 10  OR CH8_Error.ErrorPriority = 0     THEN CH8_Error.ErrorPriority := 10;     END_IF      END_IF
        IF wCH8_Diag.3  THEN    CH8_Error.sErrorMessage := CONCAT(CH8_Error.sErrorMessage, 'Short Circuit to 24V; ');       IF CH8_Error.ErrorPriority > 10  OR CH8_Error.ErrorPriority = 0     THEN CH8_Error.ErrorPriority := 10;     END_IF      END_IF
        CH8_Error.bError := TRUE;
    ELSE
        CH8_Error.bError := FALSE;
        CH8_Error.sErrorMessage := '';
    END_IF

    //Channel #9 Diag
    IF wCH9_Diag <> 0 THEN
        CH9_Error.sErrorMessage := 'EL2819 Channel #9: ';
        IF wCH9_Diag.0  THEN    CH9_Error.sErrorMessage := CONCAT(CH9_Error.sErrorMessage, 'Overtemperature; ');            IF CH9_Error.ErrorPriority > 10  OR CH9_Error.ErrorPriority = 0     THEN CH9_Error.ErrorPriority := 10;     END_IF      END_IF
        IF wCH9_Diag.1  THEN    CH9_Error.sErrorMessage := CONCAT(CH9_Error.sErrorMessage, 'Open Load; ');                  IF CH9_Error.ErrorPriority > 100 OR CH9_Error.ErrorPriority = 0     THEN CH9_Error.ErrorPriority := 100;    END_IF      END_IF
        IF wCH9_Diag.2  THEN    CH9_Error.sErrorMessage := CONCAT(CH9_Error.sErrorMessage, 'Overcurrent; ');                IF CH9_Error.ErrorPriority > 10  OR CH9_Error.ErrorPriority = 0     THEN CH9_Error.ErrorPriority := 10;     END_IF      END_IF
        IF wCH9_Diag.3  THEN    CH9_Error.sErrorMessage := CONCAT(CH9_Error.sErrorMessage, 'Short Circuit to 24V; ');       IF CH9_Error.ErrorPriority > 10  OR CH9_Error.ErrorPriority = 0     THEN CH9_Error.ErrorPriority := 10;     END_IF      END_IF
        CH9_Error.bError := TRUE;
    ELSE
        CH9_Error.bError := FALSE;
        CH9_Error.sErrorMessage := '';
    END_IF

    //Channel #10 Diag
    IF wCH10_Diag <> 0 THEN
        CH10_Error.sErrorMessage := 'EL2819 Channel #10: ';
        IF wCH10_Diag.0     THEN    CH10_Error.sErrorMessage := CONCAT(CH10_Error.sErrorMessage, 'Overtemperature; ');          IF CH10_Error.ErrorPriority > 10  OR CH10_Error.ErrorPriority = 0   THEN CH10_Error.ErrorPriority := 10;    END_IF      END_IF
        IF wCH10_Diag.1     THEN    CH10_Error.sErrorMessage := CONCAT(CH10_Error.sErrorMessage, 'Open Load; ');                IF CH10_Error.ErrorPriority > 100 OR CH10_Error.ErrorPriority = 0   THEN CH10_Error.ErrorPriority := 100;   END_IF      END_IF
        IF wCH10_Diag.2     THEN    CH10_Error.sErrorMessage := CONCAT(CH10_Error.sErrorMessage, 'Overcurrent; ');              IF CH10_Error.ErrorPriority > 10  OR CH10_Error.ErrorPriority = 0   THEN CH10_Error.ErrorPriority := 10;    END_IF      END_IF
        IF wCH10_Diag.3     THEN    CH10_Error.sErrorMessage := CONCAT(CH10_Error.sErrorMessage, 'Short Circuit to 24V; ');     IF CH10_Error.ErrorPriority > 10  OR CH10_Error.ErrorPriority = 0   THEN CH10_Error.ErrorPriority := 10;    END_IF      END_IF
        CH10_Error.bError := TRUE;
    ELSE
        CH10_Error.bError := FALSE;
        CH10_Error.sErrorMessage := '';
    END_IF

    //Channel #11 Diag
    IF wCH11_Diag <> 0 THEN
        CH11_Error.sErrorMessage := 'EL2819 Channel #11: ';
        IF wCH11_Diag.0     THEN    CH11_Error.sErrorMessage := CONCAT(CH11_Error.sErrorMessage, 'Overtemperature; ');          IF CH11_Error.ErrorPriority > 10  OR CH11_Error.ErrorPriority = 0   THEN CH11_Error.ErrorPriority := 10;    END_IF      END_IF
        IF wCH11_Diag.1     THEN    CH11_Error.sErrorMessage := CONCAT(CH11_Error.sErrorMessage, 'Open Load; ');                IF CH11_Error.ErrorPriority > 100 OR CH11_Error.ErrorPriority = 0   THEN CH11_Error.ErrorPriority := 100;   END_IF      END_IF
        IF wCH11_Diag.2     THEN    CH11_Error.sErrorMessage := CONCAT(CH11_Error.sErrorMessage, 'Overcurrent; ');              IF CH11_Error.ErrorPriority > 10  OR CH11_Error.ErrorPriority = 0   THEN CH11_Error.ErrorPriority := 10;    END_IF      END_IF
        IF wCH11_Diag.3     THEN    CH11_Error.sErrorMessage := CONCAT(CH11_Error.sErrorMessage, 'Short Circuit to 24V; ');     IF CH11_Error.ErrorPriority > 10  OR CH11_Error.ErrorPriority = 0   THEN CH11_Error.ErrorPriority := 10;    END_IF      END_IF
        CH11_Error.bError := TRUE;
    ELSE
        CH11_Error.bError := FALSE;
        CH11_Error.sErrorMessage := '';
    END_IF

    //Channel #12 Diag
    IF wCH12_Diag <> 0 THEN
        CH12_Error.sErrorMessage := 'EL2819 Channel #12: ';
        IF wCH12_Diag.0     THEN    CH12_Error.sErrorMessage := CONCAT(CH12_Error.sErrorMessage, 'Overtemperature; ');          IF CH12_Error.ErrorPriority > 10  OR CH12_Error.ErrorPriority = 0   THEN CH12_Error.ErrorPriority := 10;    END_IF      END_IF
        IF wCH12_Diag.1     THEN    CH12_Error.sErrorMessage := CONCAT(CH12_Error.sErrorMessage, 'Open Load; ');                IF CH12_Error.ErrorPriority > 100 OR CH12_Error.ErrorPriority = 0   THEN CH12_Error.ErrorPriority := 100;   END_IF      END_IF
        IF wCH12_Diag.2     THEN    CH12_Error.sErrorMessage := CONCAT(CH12_Error.sErrorMessage, 'Overcurrent; ');              IF CH12_Error.ErrorPriority > 10  OR CH12_Error.ErrorPriority = 0   THEN CH12_Error.ErrorPriority := 10;    END_IF      END_IF
        IF wCH12_Diag.3     THEN    CH12_Error.sErrorMessage := CONCAT(CH12_Error.sErrorMessage, 'Short Circuit to 24V; ');     IF CH12_Error.ErrorPriority > 10  OR CH12_Error.ErrorPriority = 0   THEN CH12_Error.ErrorPriority := 10;    END_IF      END_IF
        CH12_Error.bError := TRUE;
    ELSE
        CH12_Error.bError := FALSE;
        CH12_Error.sErrorMessage := '';
    END_IF

    //Channel #13 Diag
    IF wCH13_Diag <> 0 THEN
        CH13_Error.sErrorMessage := 'EL2819 Channel #13: ';
        IF wCH13_Diag.0     THEN    CH13_Error.sErrorMessage := CONCAT(CH13_Error.sErrorMessage, 'Overtemperature; ');          IF CH13_Error.ErrorPriority > 10  OR CH13_Error.ErrorPriority = 0   THEN CH13_Error.ErrorPriority := 10;    END_IF      END_IF
        IF wCH13_Diag.1     THEN    CH13_Error.sErrorMessage := CONCAT(CH13_Error.sErrorMessage, 'Open Load; ');                IF CH13_Error.ErrorPriority > 100 OR CH13_Error.ErrorPriority = 0   THEN CH13_Error.ErrorPriority := 100;   END_IF      END_IF
        IF wCH13_Diag.2     THEN    CH13_Error.sErrorMessage := CONCAT(CH13_Error.sErrorMessage, 'Overcurrent; ');              IF CH13_Error.ErrorPriority > 10  OR CH13_Error.ErrorPriority = 0   THEN CH13_Error.ErrorPriority := 10;    END_IF      END_IF
        IF wCH13_Diag.3     THEN    CH13_Error.sErrorMessage := CONCAT(CH13_Error.sErrorMessage, 'Short Circuit to 24V; ');     IF CH13_Error.ErrorPriority > 10  OR CH13_Error.ErrorPriority = 0   THEN CH13_Error.ErrorPriority := 10;    END_IF      END_IF
        CH13_Error.bError := TRUE;
    ELSE
        CH13_Error.bError := FALSE;
        CH13_Error.sErrorMessage := '';
    END_IF

    //Channel #14 Diag
    IF wCH14_Diag <> 0 THEN
        CH14_Error.sErrorMessage := 'EL2819 Channel #14: ';
        IF wCH14_Diag.0     THEN    CH14_Error.sErrorMessage := CONCAT(CH14_Error.sErrorMessage, 'Overtemperature; ');          IF CH14_Error.ErrorPriority > 10  OR CH14_Error.ErrorPriority = 0   THEN CH14_Error.ErrorPriority := 10;    END_IF      END_IF
        IF wCH14_Diag.1     THEN    CH14_Error.sErrorMessage := CONCAT(CH14_Error.sErrorMessage, 'Open Load; ');                IF CH14_Error.ErrorPriority > 100 OR CH14_Error.ErrorPriority = 0   THEN CH14_Error.ErrorPriority := 100;   END_IF      END_IF
        IF wCH14_Diag.2     THEN    CH14_Error.sErrorMessage := CONCAT(CH14_Error.sErrorMessage, 'Overcurrent; ');              IF CH14_Error.ErrorPriority > 10  OR CH14_Error.ErrorPriority = 0   THEN CH14_Error.ErrorPriority := 10;    END_IF      END_IF
        IF wCH14_Diag.3     THEN    CH14_Error.sErrorMessage := CONCAT(CH14_Error.sErrorMessage, 'Short Circuit to 24V; ');     IF CH14_Error.ErrorPriority > 10  OR CH14_Error.ErrorPriority = 0   THEN CH14_Error.ErrorPriority := 10;    END_IF      END_IF
        CH14_Error.bError := TRUE;
    ELSE
        CH14_Error.bError := FALSE;
        CH14_Error.sErrorMessage := '';
    END_IF

    //Channel #15 Diag
    IF wCH15_Diag <> 0 THEN
        CH15_Error.sErrorMessage := 'EL2819 Channel #15: ';
        IF wCH15_Diag.0     THEN    CH15_Error.sErrorMessage := CONCAT(CH15_Error.sErrorMessage, 'Overtemperature; ');          IF CH15_Error.ErrorPriority > 10  OR CH15_Error.ErrorPriority = 0   THEN CH15_Error.ErrorPriority := 10;    END_IF      END_IF
        IF wCH15_Diag.1     THEN    CH15_Error.sErrorMessage := CONCAT(CH15_Error.sErrorMessage, 'Open Load; ');                IF CH15_Error.ErrorPriority > 100 OR CH15_Error.ErrorPriority = 0   THEN CH15_Error.ErrorPriority := 100;   END_IF      END_IF
        IF wCH15_Diag.2     THEN    CH15_Error.sErrorMessage := CONCAT(CH15_Error.sErrorMessage, 'Overcurrent; ');              IF CH15_Error.ErrorPriority > 10  OR CH15_Error.ErrorPriority = 0   THEN CH15_Error.ErrorPriority := 10;    END_IF      END_IF
        IF wCH15_Diag.3     THEN    CH15_Error.sErrorMessage := CONCAT(CH15_Error.sErrorMessage, 'Short Circuit to 24V; ');     IF CH15_Error.ErrorPriority > 10  OR CH15_Error.ErrorPriority = 0   THEN CH15_Error.ErrorPriority := 10;    END_IF      END_IF
        CH15_Error.bError := TRUE;
    ELSE
        CH15_Error.bError := FALSE;
        CH15_Error.sErrorMessage := '';
    END_IF

    //Channel #16 Diag
    IF wCH16_Diag <> 0 THEN
        CH16_Error.sErrorMessage := 'EL2819 Channel #16: ';
        IF wCH16_Diag.0     THEN    CH16_Error.sErrorMessage := CONCAT(CH16_Error.sErrorMessage, 'Overtemperature; ');          IF CH16_Error.ErrorPriority > 10  OR CH16_Error.ErrorPriority = 0   THEN CH16_Error.ErrorPriority := 10;    END_IF      END_IF
        IF wCH16_Diag.1     THEN    CH16_Error.sErrorMessage := CONCAT(CH16_Error.sErrorMessage, 'Open Load; ');                IF CH16_Error.ErrorPriority > 100 OR CH16_Error.ErrorPriority = 0   THEN CH16_Error.ErrorPriority := 100;   END_IF      END_IF
        IF wCH16_Diag.2     THEN    CH16_Error.sErrorMessage := CONCAT(CH16_Error.sErrorMessage, 'Overcurrent; ');              IF CH16_Error.ErrorPriority > 10  OR CH16_Error.ErrorPriority = 0   THEN CH16_Error.ErrorPriority := 10;    END_IF      END_IF
        IF wCH16_Diag.3     THEN    CH16_Error.sErrorMessage := CONCAT(CH16_Error.sErrorMessage, 'Short Circuit to 24V; ');     IF CH16_Error.ErrorPriority > 10  OR CH16_Error.ErrorPriority = 0   THEN CH16_Error.ErrorPriority := 10;    END_IF      END_IF
        CH16_Error.bError := TRUE;
    ELSE
        CH16_Error.bError := FALSE;
        CH16_Error.sErrorMessage := '';
    END_IF

    //Device Diag
    IF bDev_CommonFault OR bDev_Overtemperature OR bDev_UnderVoltage OR bDev_MissingVoltage THEN
        DEV_Error.sErrorMessage := 'EL2819: ' ;
        IF bDev_CommonFault         THEN    DEV_Error.sErrorMessage := CONCAT(DEV_Error.sErrorMessage, 'Common Fault; ');               IF DEV_Error.ErrorPriority > 50  OR DEV_Error.ErrorPriority = 0 THEN DEV_Error.ErrorPriority := 50; END_IF      END_IF
        IF bDev_Overtemperature     THEN    DEV_Error.sErrorMessage := CONCAT(DEV_Error.sErrorMessage, 'Device Overtemperature; ');     IF DEV_Error.ErrorPriority > 10  OR DEV_Error.ErrorPriority = 0 THEN DEV_Error.ErrorPriority := 10; END_IF      END_IF
        IF bDev_UnderVoltage        THEN    DEV_Error.sErrorMessage := CONCAT(DEV_Error.sErrorMessage, 'Undervoltage; ');               IF DEV_Error.ErrorPriority > 10  OR DEV_Error.ErrorPriority = 0 THEN DEV_Error.ErrorPriority := 10; END_IF      END_IF
        IF bDev_MissingVoltage      THEN    DEV_Error.sErrorMessage := CONCAT(DEV_Error.sErrorMessage, 'Missing Voltage; ');            IF DEV_Error.ErrorPriority > 10  OR DEV_Error.ErrorPriority = 0 THEN DEV_Error.ErrorPriority := 10; END_IF      END_IF
        DEV_Error.bError := TRUE;
    ELSE
        DEV_Error.bError := FALSE;
        DEV_Error.sErrorMessage := '';
    END_IF

END_IF

//FB Instances
EL2819_Error(
    En                  := TRUE,
    iTerminal_ID        := iTerminal_ID,
    bWcState            := WcState_WcState,
    uiInfoData_State    := InfoData_State,
    pErrorSystem        := ErrorSystem,
    bError              => bError,
);

CH1_Error (
    En                  :=  En,
    bError              :=  ,
    sErrorMessage       :=  ,
    ErrorPriority       :=  ,
    iTerminal_ID        :=  iTerminal_ID,
    pErrorSystem        :=  ErrorSystem,
    EnO                 =>  ,
);

CH2_Error (
    En                  :=  En,
    bError              :=  ,
    sErrorMessage       :=  ,
    ErrorPriority       :=  ,
    iTerminal_ID        :=  iTerminal_ID,
    pErrorSystem        :=  ErrorSystem,
    EnO                 =>  ,
);

CH3_Error (
    En                  :=  En,
    bError              :=  ,
    sErrorMessage       :=  ,
    ErrorPriority       :=  ,
    iTerminal_ID        :=  iTerminal_ID,
    pErrorSystem        :=  ErrorSystem,
    EnO                 =>  ,
);

CH4_Error (
    En                  :=  En,
    bError              :=  ,
    sErrorMessage       :=  ,
    ErrorPriority       :=  ,
    iTerminal_ID        :=  iTerminal_ID,
    pErrorSystem        :=  ErrorSystem,
    EnO                 =>  ,
);

CH5_Error (
    En                  :=  En,
    bError              :=  ,
    sErrorMessage       :=  ,
    ErrorPriority       :=  ,
    iTerminal_ID        :=  iTerminal_ID,
    pErrorSystem        :=  ErrorSystem,
    EnO                 =>  ,
);

CH6_Error (
    En                  :=  En,
    bError              :=  ,
    sErrorMessage       :=  ,
    ErrorPriority       :=  ,
    iTerminal_ID        :=  iTerminal_ID,
    pErrorSystem        :=  ErrorSystem,
    EnO                 =>  ,
);

CH7_Error (
    En                  :=  En,
    bError              :=  ,
    sErrorMessage       :=  ,
    ErrorPriority       :=  ,
    iTerminal_ID        :=  iTerminal_ID,
    pErrorSystem        :=  ErrorSystem,
    EnO                 =>  ,
);

CH8_Error (
    En                  :=  En,
    bError              :=  ,
    sErrorMessage       :=  ,
    ErrorPriority       :=  ,
    iTerminal_ID        :=  iTerminal_ID,
    pErrorSystem        :=  ErrorSystem,
    EnO                 =>  ,
);

CH9_Error (
    En                  :=  En,
    bError              :=  ,
    sErrorMessage       :=  ,
    ErrorPriority       :=  ,
    iTerminal_ID        :=  iTerminal_ID,
    pErrorSystem        :=  ErrorSystem,
    EnO                 =>  ,
);

CH10_Error (
    En                  :=  En,
    bError              :=  ,
    sErrorMessage       :=  ,
    ErrorPriority       :=  ,
    iTerminal_ID        :=  iTerminal_ID,
    pErrorSystem        :=  ErrorSystem,
    EnO                 =>  ,
);

CH11_Error (
    En                  :=  En,
    bError              :=  ,
    sErrorMessage       :=  ,
    ErrorPriority       :=  ,
    iTerminal_ID        :=  iTerminal_ID,
    pErrorSystem        :=  ErrorSystem,
    EnO                 =>  ,
);

CH12_Error (
    En                  :=  En,
    bError              :=  ,
    sErrorMessage       :=  ,
    ErrorPriority       :=  ,
    iTerminal_ID        :=  iTerminal_ID,
    pErrorSystem        :=  ErrorSystem,
    EnO                 =>  ,
);

CH13_Error (
    En                  :=  En,
    bError              :=  ,
    sErrorMessage       :=  ,
    ErrorPriority       :=  ,
    iTerminal_ID        :=  iTerminal_ID,
    pErrorSystem        :=  ErrorSystem,
    EnO                 =>  ,
);

CH14_Error (
    En                  :=  En,
    bError              :=  ,
    sErrorMessage       :=  ,
    ErrorPriority       :=  ,
    iTerminal_ID        :=  iTerminal_ID,
    pErrorSystem        :=  ErrorSystem,
    EnO                 =>  ,
);

CH15_Error (
    En                  :=  En,
    bError              :=  ,
    sErrorMessage       :=  ,
    ErrorPriority       :=  ,
    iTerminal_ID        :=  iTerminal_ID,
    pErrorSystem        :=  ErrorSystem,
    EnO                 =>  ,
);

CH16_Error (
    En                  :=  En,
    bError              :=  ,
    sErrorMessage       :=  ,
    ErrorPriority       :=  ,
    iTerminal_ID        :=  iTerminal_ID,
    pErrorSystem        :=  ErrorSystem,
    EnO                 =>  ,
);

DEV_Error (
    En                  :=  En,
    bError              :=  ,
    sErrorMessage       :=  ,
    ErrorPriority       :=  ,
    iTerminal_ID        :=  iTerminal_ID,
    pErrorSystem        :=  ErrorSystem,
    EnO                 =>  ,
);

// Summary message
bError:=EL2819_Error.bError OR DEV_Error.bError OR CH1_Error.bError OR
CH2_Error.bError OR CH3_Error.bError OR CH4_Error.bError OR CH5_Error.bError OR
CH6_Error.bError OR CH7_Error.bError OR CH8_Error.bError OR CH9_Error.bError OR
CH10_Error.bError OR CH11_Error.bError OR CH12_Error.bError OR CH13_Error.bError OR
CH14_Error.bError OR CH15_Error.bError OR CH16_Error.bError;

IF bError THEN
  IF EL2819_Error.bError THEN
	sErrorMessage:=EL2819_Error.ErrorData.sErrorMessage;
  ELSIF DEV_Error.bError THEN
	sErrorMessage:=DEV_Error.sErrorMessage;
  ELSIF CH1_Error.bError THEN
	sErrorMessage:=CH1_Error.sErrorMessage;
  ELSIF CH2_Error.bError THEN
	sErrorMessage:=CH2_Error.sErrorMessage;
  ELSIF CH3_Error.bError THEN
	sErrorMessage:=CH3_Error.sErrorMessage;
  ELSIF CH4_Error.bError THEN
	sErrorMessage:=CH4_Error.sErrorMessage;
  ELSIF CH5_Error.bError THEN
	sErrorMessage:=CH5_Error.sErrorMessage;
  ELSIF CH6_Error.bError THEN
	sErrorMessage:=CH6_Error.sErrorMessage;
  ELSIF CH7_Error.bError THEN
	sErrorMessage:=CH7_Error.sErrorMessage;
  ELSIF CH8_Error.bError THEN
	sErrorMessage:=CH8_Error.sErrorMessage;
  ELSIF CH9_Error.bError THEN
	sErrorMessage:=CH9_Error.sErrorMessage;
  ELSIF CH10_Error.bError THEN
	sErrorMessage:=CH10_Error.sErrorMessage;
  ELSIF CH11_Error.bError THEN
	sErrorMessage:=CH11_Error.sErrorMessage;
  ELSIF CH12_Error.bError THEN
	sErrorMessage:=CH12_Error.sErrorMessage;
  ELSIF CH13_Error.bError THEN
	sErrorMessage:=CH13_Error.sErrorMessage;
  ELSIF CH14_Error.bError THEN
	sErrorMessage:=CH14_Error.sErrorMessage;
  ELSIF CH15_Error.bError THEN
	sErrorMessage:=CH15_Error.sErrorMessage;
  ELSIF CH16_Error.bError THEN
	sErrorMessage:=CH16_Error.sErrorMessage;
  ELSE
	sErrorMessage:='';
  END_IF
ELSE
  sErrorMessage:='';
END_IF

END_FUNCTION_BLOCK

// ---- POUs/Common/ErrorHandling/FB_GenericError.TcPOU
FUNCTION_BLOCK FB_GenericError

//Inputs
VAR_INPUT
    En                  : BOOL;
    bError              : BOOL;
    sErrorMessage       : STRING;
    ErrorPriority       : INT;
    iTerminal_ID        : INT;
    pErrorSystem        : POINTER TO ST_ErrorSystem;
END_VAR

//Outputs
VAR_OUTPUT
    EnO             : BOOL;
END_VAR


VAR
    LocalEntry          : ST_ErrorEntry;
    //
    sMessagePrev        : STRING;
    bMsgChanged         : BOOL;
    nErrSysCNT          :UINT;

END_VAR

(*
* ================================================================================
*                                   DESCRIPTION
* ================================================================================
* This Function Block creates a generic connection to the Error System. Unlike
* FB_TerminalError, this does not evaluate variables. Instead it checks the
* sErrorMessage & bError input variables. If bError becomes '1', a new entry is
* created in the Error System. As long as bError stays '1' every change in
* sErrorMessage inactivate the previous Error and creates a new one with the new
* message. When bError becomes '0' the last enrty is set to inactive.
* ================================================================================
*)

//Connect En to EnO
EnO := En;

IF En THEN
    //Check if pointer is OK
    IF pErrorSystem=0 THEN RETURN; END_IF

    IF sErrorMessage <> sMessagePrev THEN
        bMsgChanged := TRUE;
    ELSE
        bMsgChanged := FALSE;
    END_IF

    //Update previous value
    sMessagePrev := sErrorMessage;

    IF bMsgChanged THEN
        IF bError THEN
            IF LocalEntry.ErrorState = DUT_ErrorState.Active THEN       //Close active error
                //Read system time
                LocalEntry.sDateTimeOff := Tc2_EtherCat.DCTIME64_TO_STRING(Tc2_EtherCAT.F_GetActualDcTime64());
                LocalEntry.ErrorState   := DUT_ErrorState.Inactive;
                //Write Off-time to Error System
                FOR nErrSysCNT := 0 TO cSizeOfErrorData - 1 DO
                    IF pErrorSystem^.aErrorData[nErrSysCNT].ErrorNum = LocalEntry.ErrorNum THEN
                        pErrorSystem^.aErrorData[nErrSysCNT].sDateTimeOff   := LocalEntry.sDateTimeOff;
                        pErrorSystem^.aErrorData[nErrSysCNT].ErrorState     := DUT_ErrorState.Inactive;
                        EXIT;
                    END_IF
                END_FOR

                //Clear ErrorData
                MEMSET(ADR(LocalEntry), 0, SIZEOF(LocalEntry));
            END_IF

            //Open a new error
            LocalEntry.ErrorState       := DUT_ErrorState.Active;                                               //Set Error State
            LocalEntry.sDateTimeOn      := Tc2_EtherCat.DCTIME64_TO_STRING(Tc2_EtherCAT.F_GetActualDcTime64()); //Convert to string
            LocalEntry.sErrorMessage    := sErrorMessage;                                                       //Write message into the entry
            LocalEntry.ErrorPriority    := ErrorPriority;                                                       //Priority
            LocalEntry.iTerminalID      := iTerminal_ID;                                                        //Terminal_ID

            //Check for overflow
            IF pErrorSystem^.nNoError >= cSizeOfErrorData THEN
                pErrorSystem^.nNoOverflow   := pErrorSystem^.nNoOverflow+1;
            END_IF

            //Write Error Data into Error System
            LocalEntry.ErrorNum := pErrorSystem^.nNExtErrorNum ;
            MEMMOVE( ADR(pErrorSystem^.aErrorData[1]), ADR(pErrorSystem^.aErrorData[0]), (cSizeOfErrorData-1) * SIZEOF(ST_ErrorEntry));
            pErrorSystem^.aErrorData[0] := LocalEntry;
            pErrorSystem^.nNExtErrorNum := pErrorSystem^.nNExtErrorNum+1;

        ELSE
            //Close Active Error
            //Read system time
            LocalEntry.sDateTimeOff := Tc2_EtherCat.DCTIME64_TO_STRING(Tc2_EtherCAT.F_GetActualDcTime64());
            LocalEntry.ErrorState   := DUT_ErrorState.Inactive;

            //Write Off time to Error System
            FOR nErrSysCNT := 0 TO cSizeOfErrorData - 1 DO
                IF pErrorSystem^.aErrorData[nErrSysCNT].ErrorNum = LocalEntry.ErrorNum THEN
                    pErrorSystem^.aErrorData[nErrSysCNT].sDateTimeOff   := LocalEntry.sDateTimeOff;
                    pErrorSystem^.aErrorData[nErrSysCNT].ErrorState     := LocalEntry.ErrorState;
                    EXIT;
                END_IF
            END_FOR

            //Clear ErrorData
            MEMSET(ADR(LocalEntry), 0, SIZEOF(LocalEntry));
        END_IF
    END_IF

END_IF

END_FUNCTION_BLOCK

// ---- POUs/Common/Hardware/EtherCAT_Terminals/System/EL9505.TcPOU
//EL9505 | Power supply terminal 5V
FUNCTION_BLOCK EL9505

VAR_INPUT
    En              : BOOL;
    iTerminal_ID    : INT;
    ErrorSystem     : POINTER TO ST_ErrorSystem;
END_VAR

VAR_OUTPUT
    EnO     : BOOL;
    bError  : BOOL;
	sErrorMessage       : STRING;
END_VAR

VAR
    bUoPwr_OK           AT %I*  : BOOL;
    bUo_Overload        AT %I*  : BOOL;
    WcState_WcState     AT %I*  : BOOL;
    InfoData_State      AT %I*  : UINT;

    //FB-s
    EL9505_Error    : FB_TerminalError;
    PWR_Error       : FB_GenericError;
END_VAR

(*
* TODO: Test on hardware
*)
EnO:=En;

IF En THEN
    IF  (NOT bUoPwr_OK) OR bUo_Overload THEN
        PWR_Error.sErrorMessage     := 'EL9505: ';
        IF NOT bUoPwr_OK    THEN    PWR_Error.sErrorMessage := CONCAT (PWR_Error.sErrorMessage, 'Output Voltage Error; ');      IF PWR_Error.ErrorPriority > 5  OR PWR_Error.ErrorPriority = 0  THEN PWR_Error.ErrorPriority := 5;  END_IF  END_IF
        IF bUo_Overload     THEN    PWR_Error.sErrorMessage := CONCAT (PWR_Error.sErrorMessage, 'Overload; ');                  IF PWR_Error.ErrorPriority > 5  OR PWR_Error.ErrorPriority = 0  THEN PWR_Error.ErrorPriority := 5;  END_IF  END_IF
        PWR_Error.bError    := TRUE;
    ELSE
        PWR_Error.sErrorMessage := '';
        PWR_Error.bError        := FALSE;
    END_IF

END_IF


//Error FB instance
EL9505_Error(
    En                  := TRUE,
    iTerminal_ID        := iTerminal_ID,
    bWcState            := WcState_WcState,
    uiInfoData_State    := InfoData_State,
    pErrorSystem        := ErrorSystem,
    bError              => bError,
);

PWR_Error (
    En                  := En,
    bError              := ,
    sErrorMessage       := ,
    ErrorPriority       := ,
    iTerminal_ID        := iTerminal_ID,
    pErrorSystem        := ErrorSystem,
    EnO                 => ,
);

bError:= EL9505_Error.bError OR PWR_Error.bError;
IF bError THEN
  IF EL9505_Error.bError THEN
	sErrorMessage:=EL9505_Error.ErrorData.sErrorMessage;
  ELSIF PWR_Error.bError THEN
	sErrorMessage:=PWR_Error.sErrorMessage;
  ELSE
	sErrorMessage:='';
  END_IF
ELSE
  sErrorMessage:='';
END_IF

END_FUNCTION_BLOCK

// ---- POUs/Common/Hardware/EtherCAT_Terminals/Digital_Inputs/EL1252.TcPOU
//EL1252 or EL1252-0050 | 2-channel digitl input terminal with timestamp
FUNCTION_BLOCK EL1252
VAR_INPUT
    En              : BOOL;
    iTerminal_ID    : INT;
    ErrorSystem     : POINTER TO ST_ErrorSystem;
END_VAR

VAR_OUTPUT
    EnO     : BOOL;
    bError  : BOOL;
	sErrorMessage       : STRING;
	bBI_1                AT %I*  : BOOL:=FALSE;
	bBI_2                AT %I*  : BOOL:=FALSE;
END_VAR

VAR
    WcState_WcState     AT %I*  : BOOL;
    InfoData_State      AT %I*  : UINT;

    //FB-s
    EL1252_Error        : FB_TerminalError;
END_VAR

(*
* TODO: DONE!
*)
EnO:=En;

//Error FB instance
EL1252_Error(
    En                  := TRUE,
    iTerminal_ID        := iTerminal_ID,
    bWcState            := WcState_WcState,
    uiInfoData_State    := InfoData_State,
    pErrorSystem        := ErrorSystem,
    bError              => bError,
);

IF bError THEN
    sErrorMessage:=EL1252_Error.ErrorData.sErrorMessage;
ELSE
	sErrorMessage:='';
END_IF

END_FUNCTION_BLOCK

// ---- POUs/Common/Hardware/EtherCAT_Terminals/System/EL9410.TcPOU
//EL9410 | E-Bus power supplier and refresher, diagnostics
FUNCTION_BLOCK EL9410

VAR_INPUT
    En              : BOOL;
    iTerminal_ID    : INT;
    ErrorSystem     : POINTER TO ST_ErrorSystem;
END_VAR

VAR_OUTPUT
    EnO     : BOOL;
    bError  : BOOL;
	sErrorMessage       : STRING;
END_VAR

VAR
    bUs_Undervoltage    AT %I*  : BOOL;
    bUp_Undervoltage    AT %I*  : BOOL;
    WcState_WcState     AT %I*  : BOOL;
    InfoData_State      AT %I*  : UINT;

    //FB-s
    EL9410_Error    : FB_TerminalError;
    PWR_Error       : FB_GenericError;
END_VAR

(*
* TODO: Status bits
*)
EnO:=En;

IF En THEN
    IF  bUs_Undervoltage OR bUp_Undervoltage THEN
        PWR_Error.sErrorMessage     := 'EL9410: ';
        IF bUs_Undervoltage     THEN    PWR_Error.sErrorMessage := CONCAT (PWR_Error.sErrorMessage, 'Us undervoltage; ');       IF PWR_Error.ErrorPriority > 5  OR PWR_Error.ErrorPriority = 0  THEN PWR_Error.ErrorPriority := 5;  END_IF  END_IF
        IF bUp_Undervoltage     THEN    PWR_Error.sErrorMessage := CONCAT (PWR_Error.sErrorMessage, 'Up undervoltage; ');       IF PWR_Error.ErrorPriority > 5  OR PWR_Error.ErrorPriority = 0  THEN PWR_Error.ErrorPriority := 5;  END_IF  END_IF
        PWR_Error.bError    := TRUE;
    ELSE
        PWR_Error.sErrorMessage := '';
        PWR_Error.bError        := FALSE;
    END_IF


END_IF

//Error FB instance
EL9410_Error(
    En                  := TRUE,
    iTerminal_ID        := iTerminal_ID,
    bWcState            := WcState_WcState,
    uiInfoData_State    := InfoData_State,
    pErrorSystem        := ErrorSystem,
    bError              => bError,
);

PWR_Error (
    En                  := En,
    bError              := ,
    sErrorMessage       := ,
    ErrorPriority       := ,
    iTerminal_ID        := iTerminal_ID,
    pErrorSystem        := ErrorSystem,
    EnO                 => ,
);

bError:=EL9410_Error.bError OR PWR_Error.bError;

IF bError THEN
  IF EL9410_Error.bError THEN
	sErrorMessage:=EL9410_Error.ErrorData.sErrorMessage;
  ELSIF PWR_Error.bError THEN
	sErrorMessage:=PWR_Error.sErrorMessage;
  ELSE
	sErrorMessage:='';
  END_IF
ELSE
  sErrorMessage:='';
END_IF

END_FUNCTION_BLOCK

// ---- POUs/Common/Hardware/EtherCAT_Terminals/Feedback_Terminals/EL7201.TcPOU
//EL7201 | 1-chennel resolver terminal (ESS only use it for resolver input)
FUNCTION_BLOCK EL7201

VAR_INPUT
    En: BOOL;
    iTerminal_ID : INT;
    ErrorSystem : POINTER TO ST_ErrorSystem;
END_VAR

VAR_OUTPUT
    EnO: BOOL;
    bError: BOOL;
	sErrorMessage       : STRING;
END_VAR

VAR
    WcState_WcState AT %I* : BOOL := FALSE;
    InfoData_State  AT %I* : UINT := 0;
    fPosAct         AT %I* : UDINT := 0;
    //FB-s
    EL7201_Error    : FB_TerminalError;
END_VAR

(*
* TODO: Test on hardware
*)

EnO:=En;

EL7201_Error(
    En := TRUE,
    iTerminal_ID := iTerminal_ID,
    bWcState := FALSE,
    uiInfoData_State := InfoData_State,
    pErrorSystem := ErrorSystem,
    bError => bError,
);

IF bError THEN
	sErrorMessage:=EL7201_Error.ErrorData.sErrorMessage;
ELSE
	sErrorMessage:='';
END_IF

END_FUNCTION_BLOCK

// ---- POUs/Common/Hardware/EtherCAT_Terminals/Analog_Inputs/EL3214.TcPOU
//EL3214 | 4-channel analog input terminal, PT100 (RTD)
FUNCTION_BLOCK EL3214

VAR_INPUT
    En              : BOOL;
    iTerminal_ID    : INT;
    ErrorSystem     : POINTER TO ST_ErrorSystem;
END_VAR

VAR_OUTPUT
    EnO     : BOOL;
    bError  : BOOL;
	sErrorMessage : STRING;
	iAI_1 AT %I* :INT:=0;
	iAI_2 AT %I* :INT:=0;
	iAI_3 AT %I* :INT:=0;
	iAI_4 AT %I* :INT:=0;
END_VAR

VAR
    //Channels
    wCh1_Status     AT %I* : WORD;
    wCh2_Status     AT %I* : WORD;
    wCh3_Status     AT %I* : WORD;
    wCh4_Status     AT %I* : WORD;

    //Terminal status
    WcState_WcState     AT %I*: BOOL;
    InfoData_State      AT %I*: UINT;

    //FB-s
    EL3214_Error    : FB_TerminalError;
    CH1_Error       : FB_GenericError;
    CH2_Error       : FB_GenericError;
    CH3_Error       : FB_GenericError;
    CH4_Error       : FB_GenericError;
END_VAR

(*
* TODO: Test on hardware
*)

EnO := En;

//Channel #1 Status
IF (wCh1_Status AND 16#0043) <> 0 THEN
    CH1_Error.sErrorMessage := 'EL3214 Channel #1: ';
    IF wCh1_Status.0    THEN    CH1_Error.sErrorMessage := CONCAT(CH1_Error.sErrorMessage, 'Underrange; ');             IF CH1_Error.ErrorPriority > 100 OR CH1_Error.ErrorPriority = 0     THEN CH1_Error.ErrorPriority := 100;    END_IF      END_IF
    IF wCh1_Status.1    THEN    CH1_Error.sErrorMessage := CONCAT(CH1_Error.sErrorMessage, 'Overrange; ');              IF CH1_Error.ErrorPriority > 100 OR CH1_Error.ErrorPriority = 0     THEN CH1_Error.ErrorPriority := 100;    END_IF      END_IF
    IF wCh1_Status.6    THEN    CH1_Error.sErrorMessage := CONCAT(CH1_Error.sErrorMessage, 'Error; ');                  IF CH1_Error.ErrorPriority > 10  OR CH1_Error.ErrorPriority = 0     THEN CH1_Error.ErrorPriority := 10;     END_IF      END_IF
    CH1_Error.bError := TRUE;
ELSE
    CH1_Error.bError := FALSE;
    CH1_Error.sErrorMessage := '';
END_IF

//Channel #2 Status
IF (wCh2_Status AND 16#0043) <> 0 THEN
    CH2_Error.sErrorMessage := 'EL3214 Channel #2: ';
    IF wCh2_Status.0    THEN    CH2_Error.sErrorMessage := CONCAT(CH2_Error.sErrorMessage, 'Underrange; ');             IF CH2_Error.ErrorPriority > 100 OR CH2_Error.ErrorPriority = 0     THEN CH2_Error.ErrorPriority := 100;    END_IF      END_IF
    IF wCh2_Status.1    THEN    CH2_Error.sErrorMessage := CONCAT(CH2_Error.sErrorMessage, 'Overrange; ');              IF CH2_Error.ErrorPriority > 100 OR CH2_Error.ErrorPriority = 0     THEN CH2_Error.ErrorPriority := 100;    END_IF      END_IF
    IF wCh2_Status.6    THEN    CH2_Error.sErrorMessage := CONCAT(CH2_Error.sErrorMessage, 'Error; ');                  IF CH2_Error.ErrorPriority > 10  OR CH2_Error.ErrorPriority = 0     THEN CH2_Error.ErrorPriority := 10;     END_IF      END_IF
    CH2_Error.bError := TRUE;
ELSE
    CH2_Error.bError := FALSE;
    CH2_Error.sErrorMessage := '';
END_IF

//Channel #3 Status
IF (wCh3_Status AND 16#0043) <> 0 THEN
    CH3_Error.sErrorMessage := 'EL3214 Channel #3: ';
    IF wCh3_Status.0    THEN    CH3_Error.sErrorMessage := CONCAT(CH3_Error.sErrorMessage, 'Underrange; ');             IF CH3_Error.ErrorPriority > 100 OR CH3_Error.ErrorPriority = 0     THEN CH3_Error.ErrorPriority := 100;    END_IF      END_IF
    IF wCh3_Status.1    THEN    CH3_Error.sErrorMessage := CONCAT(CH3_Error.sErrorMessage, 'Overrange; ');              IF CH3_Error.ErrorPriority > 100 OR CH3_Error.ErrorPriority = 0     THEN CH3_Error.ErrorPriority := 100;    END_IF      END_IF
    IF wCh3_Status.6    THEN    CH3_Error.sErrorMessage := CONCAT(CH3_Error.sErrorMessage, 'Error; ');                  IF CH3_Error.ErrorPriority > 10  OR CH3_Error.ErrorPriority = 0     THEN CH3_Error.ErrorPriority := 10;     END_IF      END_IF
    CH3_Error.bError := TRUE;
ELSE
    CH3_Error.bError := FALSE;
    CH3_Error.sErrorMessage := '';
END_IF

//Channel #4 Status
IF (wCh4_Status AND 16#0043) <> 0 THEN
    CH4_Error.sErrorMessage := 'EL3214 Channel #4: ';
    IF wCh4_Status.0    THEN    CH4_Error.sErrorMessage := CONCAT(CH4_Error.sErrorMessage, 'Underrange; ');             IF CH4_Error.ErrorPriority > 100 OR CH4_Error.ErrorPriority = 0     THEN CH4_Error.ErrorPriority := 100;    END_IF      END_IF
    IF wCh4_Status.1    THEN    CH4_Error.sErrorMessage := CONCAT(CH4_Error.sErrorMessage, 'Overrange; ');              IF CH4_Error.ErrorPriority > 100 OR CH4_Error.ErrorPriority = 0     THEN CH4_Error.ErrorPriority := 100;    END_IF      END_IF
    IF wCh4_Status.6    THEN    CH4_Error.sErrorMessage := CONCAT(CH4_Error.sErrorMessage, 'Error; ');                  IF CH4_Error.ErrorPriority > 10  OR CH4_Error.ErrorPriority = 0     THEN CH4_Error.ErrorPriority := 10;     END_IF      END_IF
    CH4_Error.bError := TRUE;
ELSE
    CH4_Error.bError := FALSE;
    CH4_Error.sErrorMessage := '';
END_IF

//Error FB instance
EL3214_Error(
    En                  := TRUE,
    iTerminal_ID        := iTerminal_ID,
    bWcState            := WcState_WcState,
    uiInfoData_State    := InfoData_State,
    pErrorSystem        := ErrorSystem,
    bError              => bError,
);

CH1_Error (
    En              := En,
    bError          := ,
    sErrorMessage   := ,
    ErrorPriority   := ,
    iTerminal_ID    := iTerminal_ID,
    pErrorSystem    := ErrorSystem,
    EnO             => ,
);

CH2_Error (
    En              := En,
    bError          := ,
    sErrorMessage   := ,
    ErrorPriority   := ,
    iTerminal_ID    := iTerminal_ID,
    pErrorSystem    := ErrorSystem,
    EnO             => ,
);

CH3_Error (
    En              := En,
    bError          := ,
    sErrorMessage   := ,
    ErrorPriority   := ,
    iTerminal_ID    := iTerminal_ID,
    pErrorSystem    := ErrorSystem,
    EnO             => ,
);

CH4_Error (
    En              := En,
    bError          := ,
    sErrorMessage   := ,
    ErrorPriority   := ,
    iTerminal_ID    := iTerminal_ID,
    pErrorSystem    := ErrorSystem,
    EnO             => ,
);

bError:=EL3214_Error.bError OR CH1_Error.bError OR CH2_Error.bError OR  CH3_Error.bError OR CH4_Error.bError ;

IF bError THEN
  IF EL3214_Error.bError THEN
	sErrorMessage:=EL3214_Error.ErrorData.sErrorMessage;
  ELSIF CH1_Error.bError THEN
    sErrorMessage:=CH1_Error.sErrorMessage;
  ELSIF CH2_Error.bError THEN
    sErrorMessage:=CH2_Error.sErrorMessage;
  ELSIF CH3_Error.bError THEN
    sErrorMessage:=CH3_Error.sErrorMessage;
  ELSIF CH4_Error.bError THEN
    sErrorMessage:=CH4_Error.sErrorMessage;
  ELSE
	sErrorMessage:='';
  END_IF
ELSE 
  sErrorMessage:='';
END_IF

END_FUNCTION_BLOCK

// ---- POUs/Common/Hardware/EtherCAT_Terminals/Feedback_Terminals/EL5021.TcPOU
//EL5021 | 1-channel Sin/Cos encoder
FUNCTION_BLOCK EL5021

VAR_INPUT
    En              : BOOL;
    iTerminal_ID    : INT;
    ErrorSystem     : POINTER TO ST_ErrorSystem;
END_VAR

VAR_OUTPUT
    EnO     : BOOL;
    bError  : BOOL;
	sErrorMessage: STRING;
END_VAR

VAR
    
    InfoData_State      AT %I*  : UINT;
    WcState_WcState     AT %I*  : BOOL;
    
    //FB-s
    EL5021_Error    : FB_TerminalError;
	
END_VAR

(*
* TODO: Test on hardware
*)
EnO:=En;

